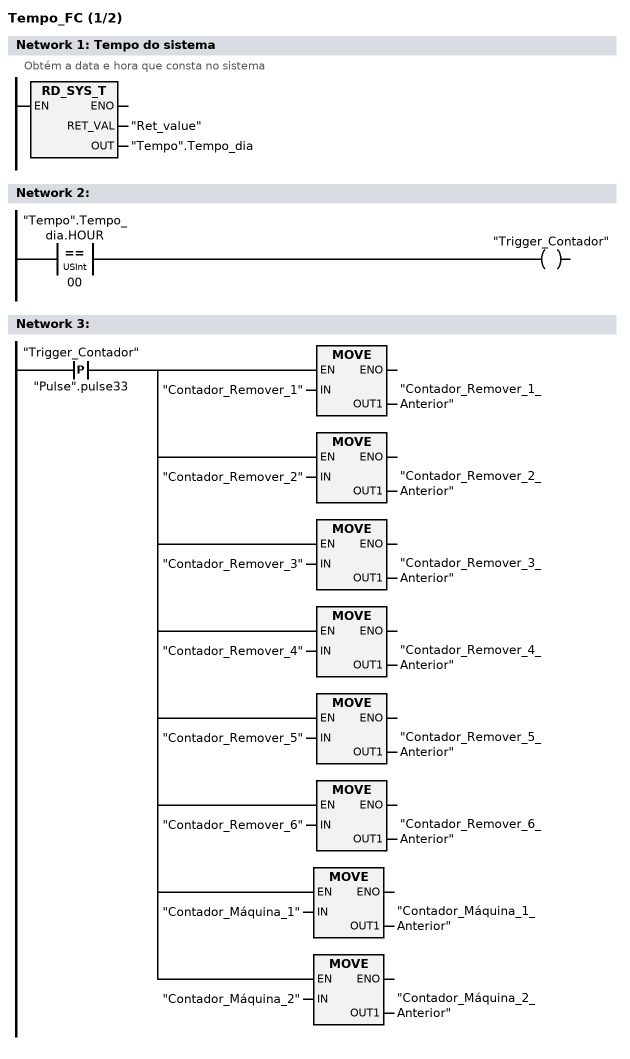
   "Ret_value" := RD_SYS_T(OUT => "Tempo".Tempo_dia);
END_REGION

REGION Network 2
   RUNG wire#powerrail
      { S7_Templates := "SrcType := USInt" } EQ_Contact(in1 := "Tempo".Tempo_dia.HOUR, in2 := 00)
      Coil( "Trigger_Contador" )
   END_RUNG
   // the same network as SCL:
   "Trigger_Contador" := "Tempo".Tempo_dia.HOUR = 00;
END_REGION

REGION Network 3
   RUNG wire#powerrail
      P_Contact(operand := "Trigger_Contador", bit := "Pulse".pulse33)
      wire#w1
      Move(in := "Contador_Remover_1", out1 => "Contador_Remover_1_Anterior")
   END_RUNG
   RUNG wire#w1
      Move(in := "Contador_Remover_2", out1 => "Contador_Remover_2_Anterior")
   END_RUNG
   RUNG wire#w1
      Move(in := "Contador_Remover_3", out1 => "Contador_Remover_3_Anterior")
   END_RUNG
   RUNG wire#w1
      Move(in := "Contador_Remover_4", out1 => "Contador_Remover_4_Anterior")
   END_RUNG
   RUNG wire#w1
      Move(in := "Contador_Remover_5", out1 => "Contador_Remover_5_Anterior")
   END_RUNG
   RUNG wire#w1
      Move(in := "Contador_Remover_6", out1 => "Contador_Remover_6_Anterior")
   END_RUNG
   RUNG wire#w1
      Move(in := "Contador_Máquina_1", out1 => "Contador_Máquina_1_Anterior")
   END_RUNG
   RUNG wire#w1
      Move(in := "Contador_Máquina_2", out1 => "Contador_Máquina_2_Anterior")
   END_RUNG
   // the same network as SCL:
   #_w1 := "Trigger_Contador" AND NOT "Pulse".pulse33;   // rising edge of "Trigger_Contador"
   "Pulse".pulse33 := "Trigger_Contador";
   IF #_w1 THEN
       "Contador_Remover_1_Anterior" := "Contador_Remover_1";
       "Contador_Remover_2_Anterior" := "Contador_Remover_2";
       "Contador_Remover_3_Anterior" := "Contador_Remover_3";
       "Contador_Remover_4_Anterior" := "Contador_Remover_4";
       "Contador_Remover_5_Anterior" := "Contador_Remover_5";
       "Contador_Remover_6_Anterior" := "Contador_Remover_6";
       "Contador_Máquina_1_Anterior" := "Contador_Máquina_1";
       "Contador_Máquina_2_Anterior" := "Contador_Máquina_2";
   END_IF;
END_REGION

REGION Network 4: Reset de contadores
   // Reset diário de todos os contadores, à meia-noite
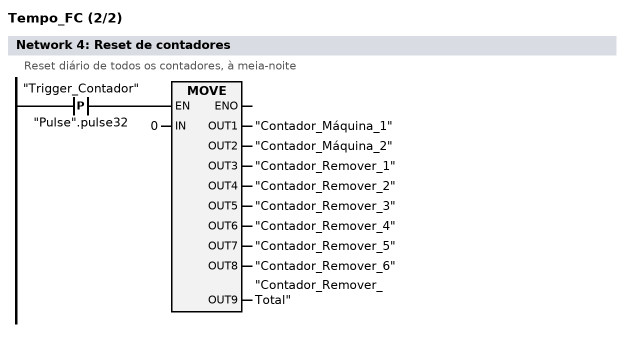
   RUNG wire#powerrail
      P_Contact(operand := "Trigger_Contador", bit := "Pulse".pulse32)
      Move(in := 0, out1 => "Contador_Máquina_1", out2 => "Contador_Máquina_2", out3 => "Contador_Remover_1", out4 => "Contador_Remover_2", out5 => "Contador_Remover_3", out6 => "Contador_Remover_4", out7 => "Contador_Remover_5", out8 => "Contador_Remover_6", out9 => "Contador_Remover_Total")
   END_RUNG
   // the same network as SCL:
   #_w1 := "Trigger_Contador" AND NOT "Pulse".pulse32;   // rising edge of "Trigger_Contador"
   "Pulse".pulse32 := "Trigger_Contador";
   IF #_w1 THEN
       "Contador_Máquina_1" := 0;
       "Contador_Máquina_2" := 0;
       "Contador_Remover_1" := 0;
       "Contador_Remover_2" := 0;
       "Contador_Remover_3" := 0;
       "Contador_Remover_4" := 0;
       "Contador_Remover_5" := 0;
       "Contador_Remover_6" := 0;
       "Contador_Remover_Total" := 0;
   END_IF;
END_REGION
END_FUNCTION

FUNCTION "MoveToSendData_PLC1" : Void   // FC10, SCL
{ S7_Optimized_Access := 'TRUE' }
VERSION : 0.1
   VAR_INPUT
      Contador_Remover_1 : DWord;
      Contador_Remover_2 : DWord;
      Contador_Remover_3 : DWord;
      Contador_Remover_4 : DWord;
      Contador_Remover_5 : DWord;
      Contador_Remover_6 : DWord;
      Contador_Remover_Total : DWord;
      Contador_Máquina_1 : DWord;
      Contador_Máquina_2 : DWord;
      "Valvula Enchimento Tanque 1" : Real;
      "Valvula Descarga Tanque 1" : Real;
      "Valvula Enchimento Tanque 2" : Real;
      "Valvula Descarga Tanque 2" : Real;
      Nivel_1_convertido_Scada : Real;
      Nivel_2_convertido_Scada : Real;
      Aviso_Nenhuma_Máquina_Habilitada : Bool;
      Aviso_Nenhum_Remover_Habilitado : Bool;
      Aviso_Sem_Condições_Empilhar : Bool;
      Set_vel_T3 : Real;
      Set_vel_T4 : Real;
      Set_vel_T5 : Real;
      Set_vel_T6 : Real;
      Set_vel_T7 : Real;
   END_VAR
   VAR_OUTPUT
      OUT_Contador_Remover_1 : DWord;
      OUT_Contador_Remover_2 : DWord;
      OUT_Contador_Remover_3 : DWord;
      OUT_Contador_Remover_4 : DWord;
      OUT_Contador_Remover_5 : DWord;
      OUT_Contador_Remover_6 : DWord;
      OUT_Contador_Remover_Total : DWord;
      OUT_Contador_Máquina_1 : DWord;
      OUT_Contador_Máquina_2 : DWord;
      "OUT_Valvula Enchimento Tanque 1" : Real;
      "OUT_Valvula Descarga Tanque 1" : Real;
      "OUT_Valvula Enchimento Tanque 2" : Real;
      "OUT_Valvula Descarga Tanque 2" : Real;
      OUT_Nivel_1_convertido_Scada : Real;
      OUT_Nivel_2_convertido_Scada : Real;
      OUT_Aviso_Nenhuma_Máquina_Habilitada : Bool;
      OUT_Aviso_Nenhum_Remover_Habilitado : Bool;
      OUT_Aviso_Sem_Condições_Empilhar : Bool;
      OUT_Set_vel_T3 : Real;
      OUT_Set_vel_T4 : Real;
      OUT_Set_vel_T5 : Real;
      OUT_Set_vel_T6 : Real;
      OUT_Set_vel_T7 : Real;
   END_VAR
BEGIN


           #OUT_Contador_Remover_1 := #Contador_Remover_1;
           #OUT_Contador_Remover_2 := #Contador_Remover_2;
           #OUT_Contador_Remover_3 := #Contador_Remover_3;
           #OUT_Contador_Remover_4 := #Contador_Remover_4;
           #OUT_Contador_Remover_5 := #Contador_Remover_5;
           #OUT_Contador_Remover_6 := #Contador_Remover_6;
           #OUT_Contador_Remover_Total := #Contador_Remover_Total;
           #OUT_Contador_Máquina_1 := #Contador_Máquina_1;
           #OUT_Contador_Máquina_2 := #Contador_Máquina_2;

           #"OUT_Valvula Enchimento Tanque 1" := #"Valvula Enchimento Tanque 1";
           #"OUT_Valvula Descarga Tanque 1":= #"Valvula Descarga Tanque 1";
           #"OUT_Valvula Enchimento Tanque 2" := #"Valvula Enchimento Tanque 2";
           #"OUT_Valvula Descarga Tanque 2":= #"Valvula Descarga Tanque 2";

           #OUT_Nivel_1_convertido_Scada := #Nivel_1_convertido_Scada;
           #OUT_Nivel_2_convertido_Scada := #Nivel_2_convertido_Scada;

           #OUT_Aviso_Nenhuma_Máquina_Habilitada := #Aviso_Nenhuma_Máquina_Habilitada;
           #OUT_Aviso_Nenhum_Remover_Habilitado := #Aviso_Nenhum_Remover_Habilitado;
           #OUT_Aviso_Sem_Condições_Empilhar := #Aviso_Sem_Condições_Empilhar;


           #OUT_Set_vel_T3 := #Set_vel_T3;
           #OUT_Set_vel_T4 := #Set_vel_T4;
           #OUT_Set_vel_T5 := #Set_vel_T5;
           #OUT_Set_vel_T6 := #Set_vel_T6;
           #OUT_Set_vel_T7 := #Set_vel_T7;
END_FUNCTION

FUNCTION "MoveToReceiveData_PLC1" : Void   // FC11, SCL
{ S7_Optimized_Access := 'TRUE' }
VERSION : 0.1
   VAR_INPUT
      Start : Bool;
      Stop : Bool;
      Emergência : Bool;
      Habilita_Remover_1 : Bool;
      Habilita_Remover_2 : Bool;
      Habilita_Remover_3 : Bool;
      Habilita_Remover_4 : Bool;
      Habilita_Remover_5 : Bool;
      Habilita_Remover_6 : Bool;
      Habilita_Máquina_1 : Bool;
      Habilita_Máquina_2 : Bool;
      Empilhar : Bool;
      Reset_Cont_Diario : DWord;
      "Reset Contadores Maquinas" : Bool;
      "Reset Contadores Postos" : Bool;
      Máquina2_Tampas : Bool;
      Máquina1_Tampas : Bool;
   END_VAR
   VAR_OUTPUT
      OUT_Start : Bool;
      OUT_Stop : Bool;
      OUT_Emergência : Bool;
      OUT_Habilita_Remover_1 : Bool;
      OUT_Habilita_Remover_2 : Bool;
      OUT_Habilita_Remover_3 : Bool;
      OUT_Habilita_Remover_4 : Bool;
      OUT_Habilita_Remover_5 : Bool;
      OUT_Habilita_Remover_6 : Bool;
      OUT_Habilita_Máquina_1 : Bool;
      OUT_Habilita_Máquina_2 : Bool;
      OUT_Empilhar : Bool;
      OUT_Reset_Cont_Diario : DWord;
      "OUT_Reset Contadores Maquinas" : Bool;
      "OUT_Reset Contadores Postos" : Bool;
      OUT_Máquina2_Tampas : Bool;
      OUT_Máquina1_Tampas : Bool;
   END_VAR
BEGIN



       #OUT_Start := #Start;
       #OUT_Stop := #Stop;
       #"OUT_Emergência" := #"Emergência";

       #OUT_Habilita_Remover_1 := #Habilita_Remover_1;
       #OUT_Habilita_Remover_2 := #Habilita_Remover_2;
       #OUT_Habilita_Remover_3 := #Habilita_Remover_3;
       #OUT_Habilita_Remover_4 := #Habilita_Remover_4;
       #OUT_Habilita_Remover_5 := #Habilita_Remover_5;
       #OUT_Habilita_Remover_6 := #Habilita_Remover_6;

       #"OUT_Habilita_Máquina_1" := #"Habilita_Máquina_1";
       #"OUT_Habilita_Máquina_2" := #"Habilita_Máquina_2";

       #OUT_Empilhar := #Empilhar;

       #OUT_Reset_Cont_Diario := #Reset_Cont_Diario;
       #"OUT_Reset Contadores Maquinas" := #"Reset Contadores Maquinas";
       #"OUT_Reset Contadores Postos" := #"Reset Contadores Postos";

       #OUT_Máquina2_Tampas := #Máquina2_Tampas;
       #OUT_Máquina1_Tampas := #Máquina1_Tampas;
END_FUNCTION

ORGANIZATION_BLOCK "Main"   // OB1, LAD, ProgramCycle
TITLE = "Main Program Sweep (Cycle)"
{ S7_Optimized_Access := 'TRUE' }
VERSION : 0.1
   VAR_INPUT
      Initial_Call : Bool;   // Initial call of this OB
      Remanence : Bool;   // =True, if remanent data are available
   END_VAR
   VAR_TEMP   // added for the SCL form of the ladder/FBD networks
      _w1 : Bool;
   END_VAR
BEGIN

REGION Network 1: Inicialização
   // Dá set ao bit do botão de stop para simular o botão de stop NC.
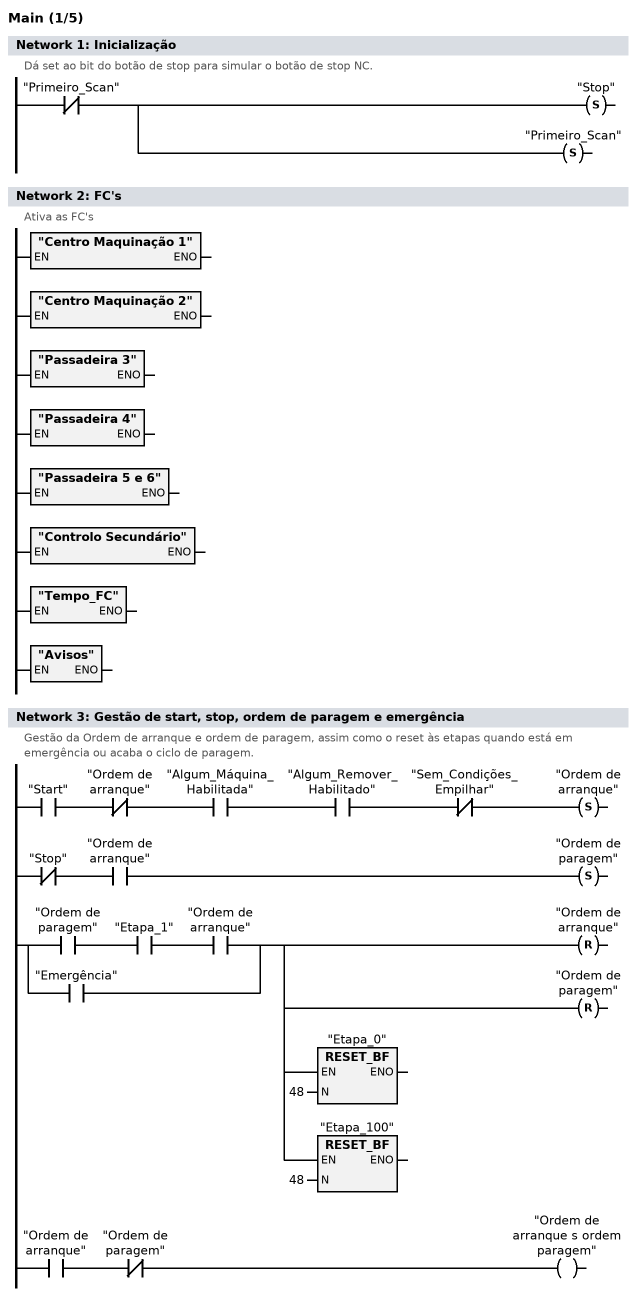
   RUNG wire#powerrail
      I_Contact( "Primeiro_Scan" )
      wire#w1
      S_Coil( "Stop" )
   END_RUNG
   RUNG wire#w1
      S_Coil( "Primeiro_Scan" )
   END_RUNG
   // the same network as SCL:
   IF NOT "Primeiro_Scan" THEN
       "Stop" := TRUE;
       "Primeiro_Scan" := TRUE;
   END_IF;
END_REGION

REGION Network 2: FC's
   // Ativa as FC's
   RUNG wire#powerrail
      "Centro Maquinação 1"()
   END_RUNG
   RUNG wire#powerrail
      "Centro Maquinação 2"()
   END_RUNG
   RUNG wire#powerrail
      "Passadeira 3"()
   END_RUNG
   RUNG wire#powerrail
      "Passadeira 4"()
   END_RUNG
   RUNG wire#powerrail
      "Passadeira 5 e 6"()
   END_RUNG
   RUNG wire#powerrail
      "Controlo Secundário"()
   END_RUNG
   RUNG wire#powerrail
      "Tempo_FC"()
   END_RUNG
   RUNG wire#powerrail
      "Avisos"()
   END_RUNG
   // the same network as SCL:
   "Centro Maquinação 1"();
   "Centro Maquinação 2"();
   "Passadeira 3"();
   "Passadeira 4"();
   "Passadeira 5 e 6"();
   "Controlo Secundário"();
   "Tempo_FC"();
   "Avisos"();
END_REGION

REGION Network 3: Gestão de start, stop, ordem de paragem e emergência
   // Gestão da Ordem de arranque e ordem de paragem, assim como o reset às etapas quando está em emergência ou acaba o ciclo de paragem.
   // no SCL statement known for RBitfield: written as a call
   IF "Start" AND NOT "Ordem de arranque" AND "Algum_Máquina_Habilitada" AND "Algum_Remover_Habilitado" AND NOT "Sem_Condições_Empilhar" THEN
       "Ordem de arranque" := TRUE;
   END_IF;
   IF NOT "Stop" AND "Ordem de arranque" THEN "Ordem de paragem" := TRUE; END_IF;
   #_w1 := ("Ordem de paragem" AND "Etapa_1" AND "Ordem de arranque") OR "Emergência";
   IF #_w1 THEN
       "Ordem de arranque" := FALSE;
       "Ordem de paragem" := FALSE;
       RESET_BF(operand := "Etapa_0", n := 48);
       RESET_BF(operand := "Etapa_100", n := 48);
   END_IF;
   "Ordem de arranque s ordem paragem" := "Ordem de arranque" AND NOT "Ordem de paragem";
END_REGION

REGION Network 4: Ordem de arranque
   // No pulse da ordem de arranque dá set à etapa 0 para iniciar
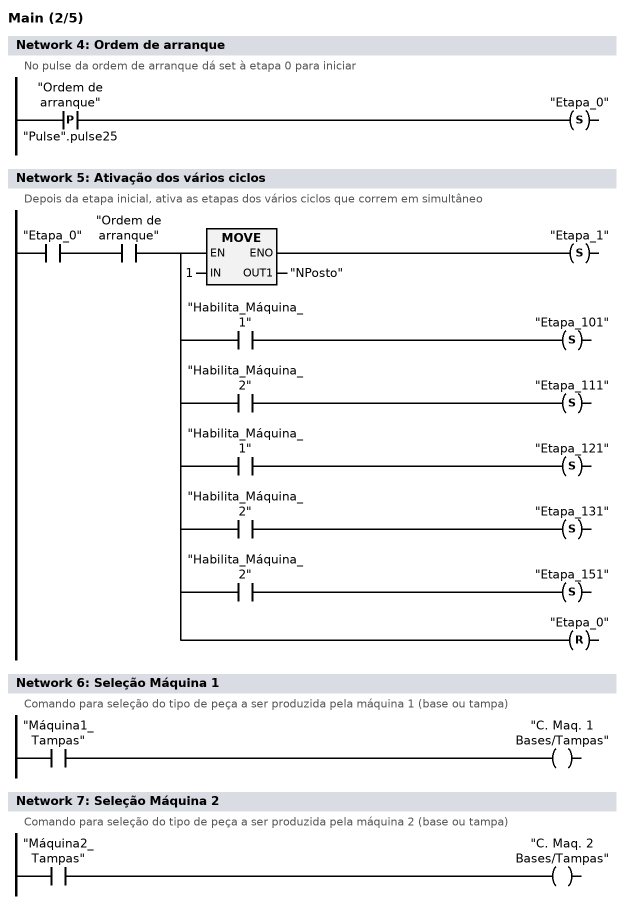
   RUNG wire#powerrail
      P_Contact(operand := "Ordem de arranque", bit := "Pulse".pulse25)
      S_Coil( "Etapa_0" )
   END_RUNG
   // the same network as SCL:
   #_w1 := "Ordem de arranque" AND NOT "Pulse".pulse25;   // rising edge of "Ordem de arranque"
   "Pulse".pulse25 := "Ordem de arranque";
   IF #_w1 THEN "Etapa_0" := TRUE; END_IF;
END_REGION

REGION Network 5: Ativação dos vários ciclos
   // Depois da etapa inicial, ativa as etapas dos vários ciclos que correm em simultâneo
   RUNG wire#powerrail
      Contact( "Etapa_0" )
      Contact( "Ordem de arranque" )
      wire#w1
      Move(in := 1, out1 => "NPosto")
      S_Coil( "Etapa_1" )
   END_RUNG
   RUNG wire#w1
      Contact( "Habilita_Máquina_1" )
      S_Coil( "Etapa_101" )
   END_RUNG
   RUNG wire#w1
      Contact( "Habilita_Máquina_2" )
      S_Coil( "Etapa_111" )
   END_RUNG
   RUNG wire#w1
      Contact( "Habilita_Máquina_1" )
      S_Coil( "Etapa_121" )
   END_RUNG
   RUNG wire#w1
      Contact( "Habilita_Máquina_2" )
      S_Coil( "Etapa_131" )
   END_RUNG
   RUNG wire#w1
      Contact( "Habilita_Máquina_2" )
      S_Coil( "Etapa_151" )
   END_RUNG
   RUNG wire#w1
      R_Coil( "Etapa_0" )
   END_RUNG
   // the same network as SCL:
   #_w1 := "Etapa_0" AND "Ordem de arranque";
   IF #_w1 THEN
       "NPosto" := 1;
       "Etapa_1" := TRUE;
   END_IF;
   IF #_w1 AND "Habilita_Máquina_1" THEN "Etapa_101" := TRUE; END_IF;
   IF #_w1 AND "Habilita_Máquina_2" THEN "Etapa_111" := TRUE; END_IF;
   IF #_w1 AND "Habilita_Máquina_1" THEN "Etapa_121" := TRUE; END_IF;
   IF #_w1 AND "Habilita_Máquina_2" THEN
       "Etapa_131" := TRUE;
       "Etapa_151" := TRUE;
   END_IF;
   IF #_w1 THEN "Etapa_0" := FALSE; END_IF;
END_REGION

REGION Network 6: Seleção Máquina 1
   // Comando para seleção do tipo de peça a ser produzida pela máquina 1 (base ou tampa)
   RUNG wire#powerrail
      Contact( "Máquina1_Tampas" )
      Coil( "C. Maq. 1 Bases/Tampas" )
   END_RUNG
   // the same network as SCL:
   "C. Maq. 1 Bases/Tampas" := "Máquina1_Tampas";
END_REGION

REGION Network 7: Seleção Máquina 2
   // Comando para seleção do tipo de peça a ser produzida pela máquina 2 (base ou tampa)
   RUNG wire#powerrail
      Contact( "Máquina2_Tampas" )
      Coil( "C. Maq. 2 Bases/Tampas" )
   END_RUNG
   // the same network as SCL:
   "C. Maq. 2 Bases/Tampas" := "Máquina2_Tampas";
END_REGION

REGION Network 8: Verificação de postos habilitados
   // Verificação de que algum posto de armazenamento está habilitado
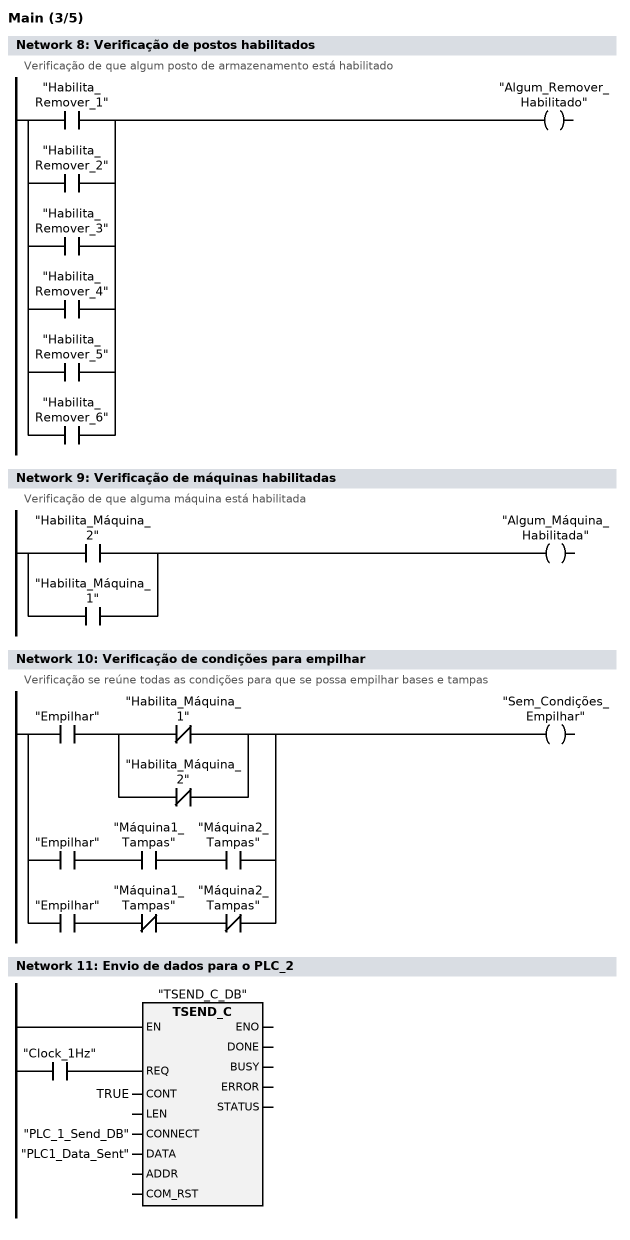
   RUNG wire#powerrail
      Contact( "Habilita_Remover_1" )
      wire#w1
      Coil( "Algum_Remover_Habilitado" )
   END_RUNG
   RUNG wire#powerrail
      Contact( "Habilita_Remover_2" )
   END_RUNG wire#w1
   RUNG wire#powerrail
      Contact( "Habilita_Remover_3" )
   END_RUNG wire#w1
   RUNG wire#powerrail
      Contact( "Habilita_Remover_4" )
   END_RUNG wire#w1
   RUNG wire#powerrail
      Contact( "Habilita_Remover_5" )
   END_RUNG wire#w1
   RUNG wire#powerrail
      Contact( "Habilita_Remover_6" )
   END_RUNG wire#w1
   // the same network as SCL:
   "Algum_Remover_Habilitado" := "Habilita_Remover_1" OR "Habilita_Remover_2" OR "Habilita_Remover_3" OR "Habilita_Remover_4" OR "Habilita_Remover_5" OR "Habilita_Remover_6";
END_REGION

REGION Network 9: Verificação de máquinas habilitadas
   // Verificação de que alguma máquina está habilitada
   RUNG wire#powerrail
      Contact( "Habilita_Máquina_2" )
      wire#w1
      Coil( "Algum_Máquina_Habilitada" )
   END_RUNG
   RUNG wire#powerrail
      Contact( "Habilita_Máquina_1" )
   END_RUNG wire#w1
   // the same network as SCL:
   "Algum_Máquina_Habilitada" := "Habilita_Máquina_2" OR "Habilita_Máquina_1";
END_REGION

REGION Network 10: Verificação de condições para empilhar
   // Verificação se reúne todas as condições para que se possa empilhar bases e tampas
   RUNG wire#powerrail
      Contact( "Empilhar" )
      wire#w1
      I_Contact( "Habilita_Máquina_1" )
      wire#w2
      Coil( "Sem_Condições_Empilhar" )
   END_RUNG
   RUNG wire#w1
      I_Contact( "Habilita_Máquina_2" )
   END_RUNG wire#w2
   RUNG wire#powerrail
      Contact( "Empilhar" )
      Contact( "Máquina1_Tampas" )
      Contact( "Máquina2_Tampas" )
   END_RUNG wire#w2
   RUNG wire#powerrail
      Contact( "Empilhar" )
      I_Contact( "Máquina1_Tampas" )
      I_Contact( "Máquina2_Tampas" )
   END_RUNG wire#w2
   // the same network as SCL:
   "Sem_Condições_Empilhar" := ("Empilhar" AND (NOT "Habilita_Máquina_1" OR NOT "Habilita_Máquina_2")) OR ("Empilhar" AND "Máquina1_Tampas" AND "Máquina2_Tampas") OR ("Empilhar" AND NOT "Máquina1_Tampas" AND NOT "Máquina2_Tampas");
END_REGION

REGION Network 11: Envio de dados para o PLC_2
   "TSEND_C_DB"(REQ := "Clock_1Hz", CONT := TRUE, CONNECT := "PLC_1_Send_DB", DATA := "PLC1_Data_Sent");   // TSEND_C
END_REGION

REGION Network 12: Função para copiar os valores das variáveis para uma DB que partilhará os dados com o PLC_2
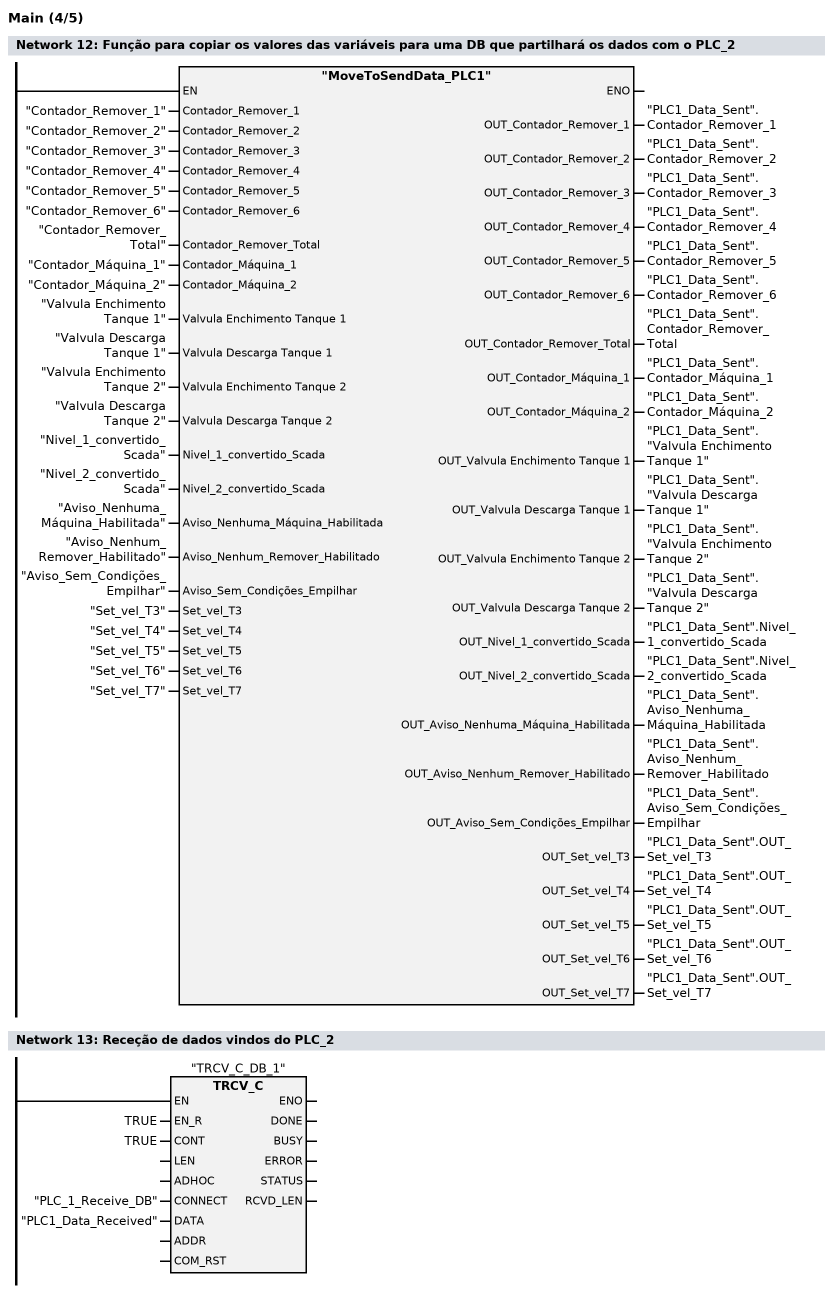
   RUNG wire#powerrail
      "MoveToSendData_PLC1"(Contador_Remover_1 := "Contador_Remover_1", Contador_Remover_2 := "Contador_Remover_2", Contador_Remover_3 := "Contador_Remover_3", Contador_Remover_4 := "Contador_Remover_4", Contador_Remover_5 := "Contador_Remover_5", Contador_Remover_6 := "Contador_Remover_6", Contador_Remover_Total := "Contador_Remover_Total", Contador_Máquina_1 := "Contador_Máquina_1", Contador_Máquina_2 := "Contador_Máquina_2", "Valvula Enchimento Tanque 1" := "Valvula Enchimento Tanque 1", "Valvula Descarga Tanque 1" := "Valvula Descarga Tanque 1", "Valvula Enchimento Tanque 2" := "Valvula Enchimento Tanque 2", "Valvula Descarga Tanque 2" := "Valvula Descarga Tanque 2", Nivel_1_convertido_Scada := "Nivel_1_convertido_Scada", Nivel_2_convertido_Scada := "Nivel_2_convertido_Scada", Aviso_Nenhuma_Máquina_Habilitada := "Aviso_Nenhuma_Máquina_Habilitada", Aviso_Nenhum_Remover_Habilitado := "Aviso_Nenhum_Remover_Habilitado", Aviso_Sem_Condições_Empilhar := "Aviso_Sem_Condições_Empilhar", Set_vel_T3 := "Set_vel_T3", Set_vel_T4 := "Set_vel_T4", Set_vel_T5 := "Set_vel_T5", Set_vel_T6 := "Set_vel_T6", Set_vel_T7 := "Set_vel_T7", OUT_Contador_Remover_1 => "PLC1_Data_Sent".Contador_Remover_1, OUT_Contador_Remover_2 => "PLC1_Data_Sent".Contador_Remover_2, OUT_Contador_Remover_3 => "PLC1_Data_Sent".Contador_Remover_3, OUT_Contador_Remover_4 => "PLC1_Data_Sent".Contador_Remover_4, OUT_Contador_Remover_5 => "PLC1_Data_Sent".Contador_Remover_5, OUT_Contador_Remover_6 => "PLC1_Data_Sent".Contador_Remover_6, OUT_Contador_Remover_Total => "PLC1_Data_Sent".Contador_Remover_Total, OUT_Contador_Máquina_1 => "PLC1_Data_Sent".Contador_Máquina_1, OUT_Contador_Máquina_2 => "PLC1_Data_Sent".Contador_Máquina_2, "OUT_Valvula Enchimento Tanque 1" => "PLC1_Data_Sent"."Valvula Enchimento Tanque 1", "OUT_Valvula Descarga Tanque 1" => "PLC1_Data_Sent"."Valvula Descarga Tanque 1", "OUT_Valvula Enchimento Tanque 2" => "PLC1_Data_Sent"."Valvula Enchimento Tanque 2", "OUT_Valvula Descarga Tanque 2" => "PLC1_Data_Sent"."Valvula Descarga Tanque 2", OUT_Nivel_1_convertido_Scada => "PLC1_Data_Sent".Nivel_1_convertido_Scada, OUT_Nivel_2_convertido_Scada => "PLC1_Data_Sent".Nivel_2_convertido_Scada, OUT_Aviso_Nenhuma_Máquina_Habilitada => "PLC1_Data_Sent".Aviso_Nenhuma_Máquina_Habilitada, OUT_Aviso_Nenhum_Remover_Habilitado => "PLC1_Data_Sent".Aviso_Nenhum_Remover_Habilitado, OUT_Aviso_Sem_Condições_Empilhar => "PLC1_Data_Sent".Aviso_Sem_Condições_Empilhar, OUT_Set_vel_T3 => "PLC1_Data_Sent".OUT_Set_vel_T3, OUT_Set_vel_T4 => "PLC1_Data_Sent".OUT_Set_vel_T4, OUT_Set_vel_T5 => "PLC1_Data_Sent".OUT_Set_vel_T5, OUT_Set_vel_T6 => "PLC1_Data_Sent".OUT_Set_vel_T6, OUT_Set_vel_T7 => "PLC1_Data_Sent".OUT_Set_vel_T7)
   END_RUNG
   // the same network as SCL:
   "MoveToSendData_PLC1"(Contador_Remover_1 := "Contador_Remover_1",
                         Contador_Remover_2 := "Contador_Remover_2",
                         Contador_Remover_3 := "Contador_Remover_3",
                         Contador_Remover_4 := "Contador_Remover_4",
                         Contador_Remover_5 := "Contador_Remover_5",
                         Contador_Remover_6 := "Contador_Remover_6",
                         Contador_Remover_Total := "Contador_Remover_Total",
                         Contador_Máquina_1 := "Contador_Máquina_1",
                         Contador_Máquina_2 := "Contador_Máquina_2",
                         "Valvula Enchimento Tanque 1" := "Valvula Enchimento Tanque 1",
                         "Valvula Descarga Tanque 1" := "Valvula Descarga Tanque 1",
                         "Valvula Enchimento Tanque 2" := "Valvula Enchimento Tanque 2",
                         "Valvula Descarga Tanque 2" := "Valvula Descarga Tanque 2",
                         Nivel_1_convertido_Scada := "Nivel_1_convertido_Scada",
                         Nivel_2_convertido_Scada := "Nivel_2_convertido_Scada",
                         Aviso_Nenhuma_Máquina_Habilitada := "Aviso_Nenhuma_Máquina_Habilitada",
                         Aviso_Nenhum_Remover_Habilitado := "Aviso_Nenhum_Remover_Habilitado",
                         Aviso_Sem_Condições_Empilhar := "Aviso_Sem_Condições_Empilhar",
                         Set_vel_T3 := "Set_vel_T3",
                         Set_vel_T4 := "Set_vel_T4",
                         Set_vel_T5 := "Set_vel_T5",
                         Set_vel_T6 := "Set_vel_T6",
                         Set_vel_T7 := "Set_vel_T7",
                         OUT_Contador_Remover_1 => "PLC1_Data_Sent".Contador_Remover_1,
                         OUT_Contador_Remover_2 => "PLC1_Data_Sent".Contador_Remover_2,
                         OUT_Contador_Remover_3 => "PLC1_Data_Sent".Contador_Remover_3,
                         OUT_Contador_Remover_4 => "PLC1_Data_Sent".Contador_Remover_4,
                         OUT_Contador_Remover_5 => "PLC1_Data_Sent".Contador_Remover_5,
                         OUT_Contador_Remover_6 => "PLC1_Data_Sent".Contador_Remover_6,
                         OUT_Contador_Remover_Total => "PLC1_Data_Sent".Contador_Remover_Total,
                         OUT_Contador_Máquina_1 => "PLC1_Data_Sent".Contador_Máquina_1,
                         OUT_Contador_Máquina_2 => "PLC1_Data_Sent".Contador_Máquina_2,
                         "OUT_Valvula Enchimento Tanque 1" => "PLC1_Data_Sent"."Valvula Enchimento Tanque 1",
                         "OUT_Valvula Descarga Tanque 1" => "PLC1_Data_Sent"."Valvula Descarga Tanque 1",
                         "OUT_Valvula Enchimento Tanque 2" => "PLC1_Data_Sent"."Valvula Enchimento Tanque 2",
                         "OUT_Valvula Descarga Tanque 2" => "PLC1_Data_Sent"."Valvula Descarga Tanque 2",
                         OUT_Nivel_1_convertido_Scada => "PLC1_Data_Sent".Nivel_1_convertido_Scada,
                         OUT_Nivel_2_convertido_Scada => "PLC1_Data_Sent".Nivel_2_convertido_Scada,
                         OUT_Aviso_Nenhuma_Máquina_Habilitada => "PLC1_Data_Sent".Aviso_Nenhuma_Máquina_Habilitada,
                         OUT_Aviso_Nenhum_Remover_Habilitado => "PLC1_Data_Sent".Aviso_Nenhum_Remover_Habilitado,
                         OUT_Aviso_Sem_Condições_Empilhar => "PLC1_Data_Sent".Aviso_Sem_Condições_Empilhar,
                         OUT_Set_vel_T3 => "PLC1_Data_Sent".OUT_Set_vel_T3,
                         OUT_Set_vel_T4 => "PLC1_Data_Sent".OUT_Set_vel_T4,
                         OUT_Set_vel_T5 => "PLC1_Data_Sent".OUT_Set_vel_T5,
                         OUT_Set_vel_T6 => "PLC1_Data_Sent".OUT_Set_vel_T6,
                         OUT_Set_vel_T7 => "PLC1_Data_Sent".OUT_Set_vel_T7);
END_REGION

REGION Network 13: Receção de dados vindos do PLC_2
   "TRCV_C_DB_1"(EN_R := TRUE, CONT := TRUE, CONNECT := "PLC_1_Receive_DB", DATA := "PLC1_Data_Received");   // TRCV_C
END_REGION

REGION Network 14
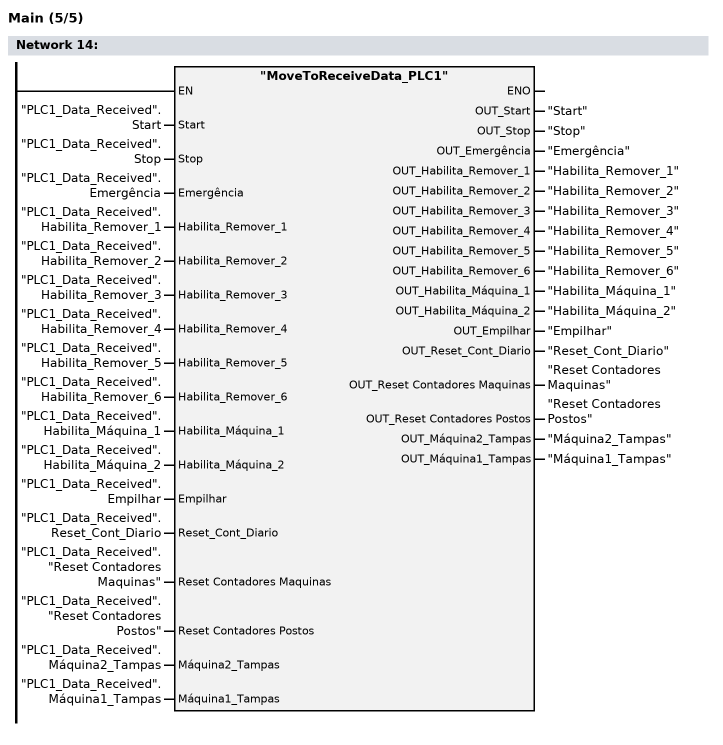
   RUNG wire#powerrail
      "MoveToReceiveData_PLC1"(Start := "PLC1_Data_Received".Start, Stop := "PLC1_Data_Received".Stop, Emergência := "PLC1_Data_Received".Emergência, Habilita_Remover_1 := "PLC1_Data_Received".Habilita_Remover_1, Habilita_Remover_2 := "PLC1_Data_Received".Habilita_Remover_2, Habilita_Remover_3 := "PLC1_Data_Received".Habilita_Remover_3, Habilita_Remover_4 := "PLC1_Data_Received".Habilita_Remover_4, Habilita_Remover_5 := "PLC1_Data_Received".Habilita_Remover_5, Habilita_Remover_6 := "PLC1_Data_Received".Habilita_Remover_6, Habilita_Máquina_1 := "PLC1_Data_Received".Habilita_Máquina_1, Habilita_Máquina_2 := "PLC1_Data_Received".Habilita_Máquina_2, Empilhar := "PLC1_Data_Received".Empilhar, Reset_Cont_Diario := "PLC1_Data_Received".Reset_Cont_Diario, "Reset Contadores Maquinas" := "PLC1_Data_Received"."Reset Contadores Maquinas", "Reset Contadores Postos" := "PLC1_Data_Received"."Reset Contadores Postos", Máquina2_Tampas := "PLC1_Data_Received".Máquina2_Tampas, Máquina1_Tampas := "PLC1_Data_Received".Máquina1_Tampas, OUT_Start => "Start", OUT_Stop => "Stop", OUT_Emergência => "Emergência", OUT_Habilita_Remover_1 => "Habilita_Remover_1", OUT_Habilita_Remover_2 => "Habilita_Remover_2", OUT_Habilita_Remover_3 => "Habilita_Remover_3", OUT_Habilita_Remover_4 => "Habilita_Remover_4", OUT_Habilita_Remover_5 => "Habilita_Remover_5", OUT_Habilita_Remover_6 => "Habilita_Remover_6", OUT_Habilita_Máquina_1 => "Habilita_Máquina_1", OUT_Habilita_Máquina_2 => "Habilita_Máquina_2", OUT_Empilhar => "Empilhar", OUT_Reset_Cont_Diario => "Reset_Cont_Diario", "OUT_Reset Contadores Maquinas" => "Reset Contadores Maquinas", "OUT_Reset Contadores Postos" => "Reset Contadores Postos", OUT_Máquina2_Tampas => "Máquina2_Tampas", OUT_Máquina1_Tampas => "Máquina1_Tampas")
   END_RUNG
   // the same network as SCL:
   "MoveToReceiveData_PLC1"(Start := "PLC1_Data_Received".Start,
                           Stop := "PLC1_Data_Received".Stop,
                           Emergência := "PLC1_Data_Received".Emergência,
                           Habilita_Remover_1 := "PLC1_Data_Received".Habilita_Remover_1,
                           Habilita_Remover_2 := "PLC1_Data_Received".Habilita_Remover_2,
                           Habilita_Remover_3 := "PLC1_Data_Received".Habilita_Remover_3,
                           Habilita_Remover_4 := "PLC1_Data_Received".Habilita_Remover_4,
                           Habilita_Remover_5 := "PLC1_Data_Received".Habilita_Remover_5,
                           Habilita_Remover_6 := "PLC1_Data_Received".Habilita_Remover_6,
                           Habilita_Máquina_1 := "PLC1_Data_Received".Habilita_Máquina_1,
                           Habilita_Máquina_2 := "PLC1_Data_Received".Habilita_Máquina_2,
                           Empilhar := "PLC1_Data_Received".Empilhar,
                           Reset_Cont_Diario := "PLC1_Data_Received".Reset_Cont_Diario,
                           "Reset Contadores Maquinas" := "PLC1_Data_Received"."Reset Contadores Maquinas",
                           "Reset Contadores Postos" := "PLC1_Data_Received"."Reset Contadores Postos",
                           Máquina2_Tampas := "PLC1_Data_Received".Máquina2_Tampas,
                           Máquina1_Tampas := "PLC1_Data_Received".Máquina1_Tampas,
                           OUT_Start => "Start",
                           OUT_Stop => "Stop",
                           OUT_Emergência => "Emergência",
                           OUT_Habilita_Remover_1 => "Habilita_Remover_1",
                           OUT_Habilita_Remover_2 => "Habilita_Remover_2",
                           OUT_Habilita_Remover_3 => "Habilita_Remover_3",
                           OUT_Habilita_Remover_4 => "Habilita_Remover_4",
                           OUT_Habilita_Remover_5 => "Habilita_Remover_5",
                           OUT_Habilita_Remover_6 => "Habilita_Remover_6",
                           OUT_Habilita_Máquina_1 => "Habilita_Máquina_1",
                           OUT_Habilita_Máquina_2 => "Habilita_Máquina_2",
                           OUT_Empilhar => "Empilhar",
                           OUT_Reset_Cont_Diario => "Reset_Cont_Diario",
                           "OUT_Reset Contadores Maquinas" => "Reset Contadores Maquinas",
                           "OUT_Reset Contadores Postos" => "Reset Contadores Postos",
                           OUT_Máquina2_Tampas => "Máquina2_Tampas",
                           OUT_Máquina1_Tampas => "Máquina1_Tampas");
END_REGION
END_ORGANIZATION_BLOCK

ORGANIZATION_BLOCK "Cyclic interrupt"   // OB30, LAD, CyclicInterrupt
TITLE = PID Tanque 1
{ S7_Optimized_Access := 'TRUE' }
VERSION : 0.1
   VAR_INPUT
      Initial_Call : Bool;   // Initial call of this OB
      Event_Count : Int;   // Events discarded
   END_VAR
   VAR_TEMP
      erro : Int;
   END_VAR
BEGIN

REGION Network 1: PID do Tanque 1
   // Definição do PID do Tanque 1
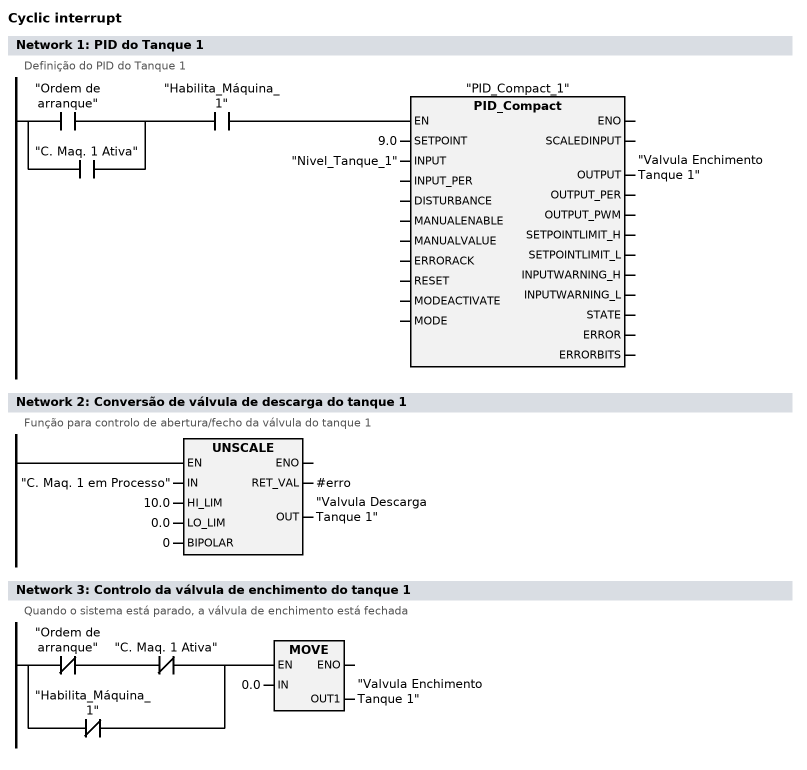
   IF ("Ordem de arranque" OR "C. Maq. 1 Ativa") AND "Habilita_Máquina_1" THEN
       "PID_Compact_1"(Setpoint := 9.0, Input := "Nivel_Tanque_1", Output => "Valvula Enchimento Tanque 1");   // PID_Compact
   END_IF;
END_REGION

REGION Network 2: Conversão de válvula de descarga do tanque 1
   // Função para controlo de abertura/fecho da válvula do tanque 1
   #erro := UNSCALE(IN := "C. Maq. 1 em Processo",
                    HI_LIM := 10.0,
                    LO_LIM := 0.0,
                    BIPOLAR := 0,
                    OUT => "Valvula Descarga Tanque 1");
END_REGION

REGION Network 3: Controlo da válvula de enchimento do tanque 1
   // Quando o sistema está parado, a válvula de enchimento está fechada
   RUNG wire#powerrail
      I_Contact( "Ordem de arranque" )
      I_Contact( "C. Maq. 1 Ativa" )
      wire#w1
      Move(in := 0.0, out1 => "Valvula Enchimento Tanque 1")
   END_RUNG
   RUNG wire#powerrail
      I_Contact( "Habilita_Máquina_1" )
   END_RUNG wire#w1
   // the same network as SCL:
   IF (NOT "Ordem de arranque" AND NOT "C. Maq. 1 Ativa") OR NOT "Habilita_Máquina_1" THEN
       "Valvula Enchimento Tanque 1" := 0.0;
   END_IF;
END_REGION
END_ORGANIZATION_BLOCK

ORGANIZATION_BLOCK "Cyclic interrupt_1"   // OB31, LAD, CyclicInterrupt
TITLE = PID Tanque 2
{ S7_Optimized_Access := 'TRUE' }
VERSION : 0.1
   VAR_INPUT
      Initial_Call : Bool;   // Initial call of this OB
      Event_Count : Int;   // Events discarded
   END_VAR
   VAR_TEMP
      erro : Int;
   END_VAR
BEGIN

REGION Network 1: PID do Tanque 2
   // Definição do PID do Tanque 2
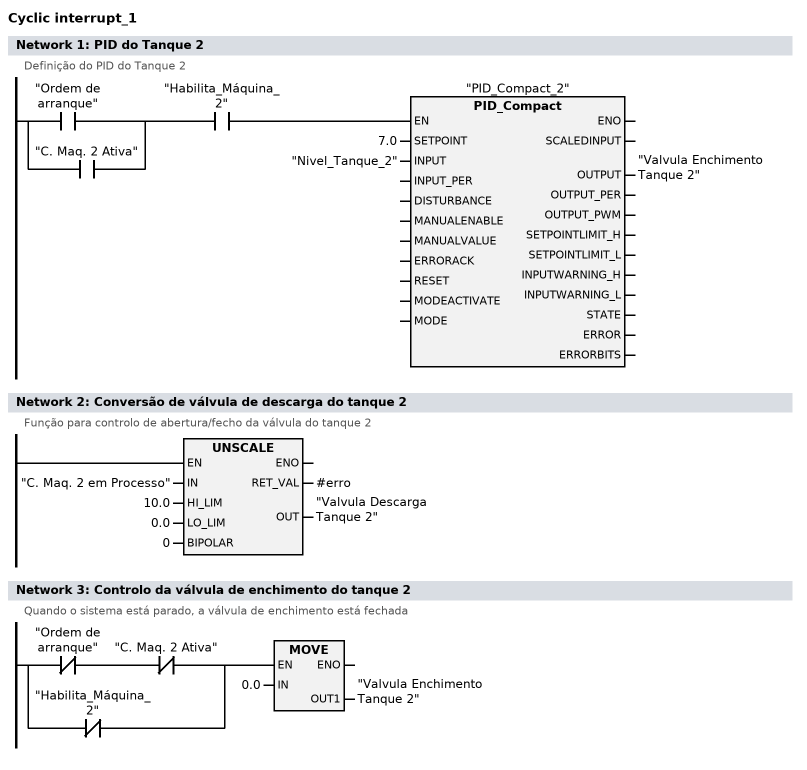
   IF ("Ordem de arranque" OR "C. Maq. 2 Ativa") AND "Habilita_Máquina_2" THEN
       "PID_Compact_2"(Setpoint := 7.0, Input := "Nivel_Tanque_2", Output => "Valvula Enchimento Tanque 2");   // PID_Compact
   END_IF;
END_REGION

REGION Network 2: Conversão de válvula de descarga do tanque 2
   // Função para controlo de abertura/fecho da válvula do tanque 2
   #erro := UNSCALE(IN := "C. Maq. 2 em Processo",
                    HI_LIM := 10.0,
                    LO_LIM := 0.0,
                    BIPOLAR := 0,
                    OUT => "Valvula Descarga Tanque 2");
END_REGION

REGION Network 3: Controlo da válvula de enchimento do tanque 2
   // Quando o sistema está parado, a válvula de enchimento está fechada
   RUNG wire#powerrail
      I_Contact( "Ordem de arranque" )
      I_Contact( "C. Maq. 2 Ativa" )
      wire#w1
      Move(in := 0.0, out1 => "Valvula Enchimento Tanque 2")
   END_RUNG
   RUNG wire#powerrail
      I_Contact( "Habilita_Máquina_2" )
   END_RUNG wire#w1
   // the same network as SCL:
   IF (NOT "Ordem de arranque" AND NOT "C. Maq. 2 Ativa") OR NOT "Habilita_Máquina_2" THEN
       "Valvula Enchimento Tanque 2" := 0.0;
   END_IF;
END_REGION
END_ORGANIZATION_BLOCK

// ===== PLC "PLC_2"  CPU 1512C-1 PN =====

VAR_GLOBAL   // PLC tag table "Default tag table"
   "Clock_Byte" AT %MB500 : Byte;
   "Clock_10Hz" AT %M500.0 : Bool;
   "Clock_5Hz" AT %M500.1 : Bool;
   "Clock_2.5Hz" AT %M500.2 : Bool;
   "Clock_2Hz" AT %M500.3 : Bool;
   "Clock_1.25Hz" AT %M500.4 : Bool;
   "Clock_1Hz" AT %M500.5 : Bool;
   "Clock_0.625Hz" AT %M500.6 : Bool;
   "Clock_0.5Hz" AT %M500.7 : Bool;
END_VAR

DATA_BLOCK "PLC2_Data_Received"   // DB3
{ S7_Optimized_Access := 'FALSE' }
VERSION : 0.1
   VAR
      Contador_Remover_1 : DWord;
      Contador_Remover_2 : DWord;
      Contador_Remover_3 : DWord;
      Contador_Remover_4 : DWord;
      Contador_Remover_5 : DWord;
      Contador_Remover_6 : DWord;
      Contador_Remover_Total : DWord;
      Contador_Máquina_1 : DWord;
      Contador_Máquina_2 : DWord;
      "Valvula Enchimento Tanque 1" : Real;
      "Valvula Descarga Tanque 1" : Real;
      "Valvula Enchimento Tanque 2" : Real;
      "Valvula Descarga Tanque 2" : Real;
      Nivel_1_convertido_Scada : Real;
      Nivel_2_convertido_Scada : Real;
      Aviso_Nenhuma_Máquina_Habilitada : Bool;
      Aviso_Nenhum_Remover_Habilitado : Bool;
      Aviso_Sem_Condições_Empilhar : Bool;
      Set_vel_T3 : Real;
      Set_vel_T4 : Real;
      Set_vel_T6 : Real;
      Set_vel_T5 : Real;
      Set_vel_T7 : Real;
   END_VAR
BEGIN
END_DATA_BLOCK

DATA_BLOCK "PLC2_Data_Sent"   // DB5
{ S7_Optimized_Access := 'FALSE' }
VERSION : 0.1
   VAR
      Start : Bool;
      Stop : Bool;
      Emergência : Bool;
      Habilita_Remover_1 : Bool;
      Habilita_Remover_2 : Bool;
      Habilita_Remover_3 : Bool;
      Habilita_Remover_4 : Bool;
      Habilita_Remover_5 : Bool;
      Habilita_Remover_6 : Bool;
      Habilita_Máquina_1 : Bool;
      Habilita_Máquina_2 : Bool;
      Empilhar : Bool;
      Reset_Cont_Diario : Bool;
      "Reset Contadores Maquinas" : Bool;
      "Reset Contadores Postos" : Bool;
      Máquina1_Tampas : Bool;
      Máquina2_Tampas : Bool;
   END_VAR
BEGIN
END_DATA_BLOCK

// folder: System blocks/Program resources

DATA_BLOCK "PLC_2_Receive_DB"   // DB1
{ S7_Optimized_Access := 'TRUE' }
AUTHOR : SIMATIC
FAMILY : MC7Plus
NAME : TC_IP_v4
VERSION : 1.0
// stored: InstanceOfName TCON_IP_v4
"TCON_IP_v4"
BEGIN
   ID := 1;
   InterfaceId := 64;
   LocalPort := 2000;
   RemoteAddress.ADDR[1] := 192;
   RemoteAddress.ADDR[2] := 168;
   RemoteAddress.ADDR[3] := 228;
   RemoteAddress.ADDR[4] := 231;
END_DATA_BLOCK

DATA_BLOCK "PLC_2_Send_DB"   // DB6
{ S7_Optimized_Access := 'TRUE' }
AUTHOR : SIMATIC
FAMILY : MC7Plus
NAME : TC_IP_v4
VERSION : 1.0
// stored: InstanceOfName TCON_IP_v4
"TCON_IP_v4"
BEGIN
   ID := 2;
   InterfaceId := 64;
   RemotePort := 2000;
   ActiveEstablished := true;
   RemoteAddress.ADDR[1] := 192;
   RemoteAddress.ADDR[2] := 168;
   RemoteAddress.ADDR[3] := 228;
   RemoteAddress.ADDR[4] := 231;
END_DATA_BLOCK

// folder: (top level)

ORGANIZATION_BLOCK "Main"   // OB1, LAD, ProgramCycle
TITLE = "Main Program Sweep (Cycle)"
{ S7_Optimized_Access := 'TRUE' }
VERSION : 0.1
   VAR_INPUT
      Initial_Call : Bool;   // Initial call of this OB
      Remanence : Bool;   // =True, if remanent data are available
   END_VAR
BEGIN

REGION Network 1
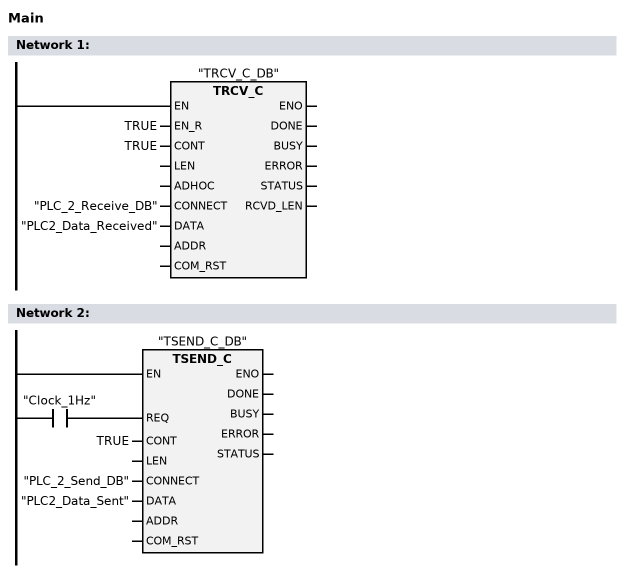
   "TRCV_C_DB"(EN_R := TRUE, CONT := TRUE, CONNECT := "PLC_2_Receive_DB", DATA := "PLC2_Data_Received");   // TRCV_C
END_REGION

REGION Network 2
   "TSEND_C_DB"(REQ := "Clock_1Hz", CONT := TRUE, CONNECT := "PLC_2_Send_DB", DATA := "PLC2_Data_Sent");   // TSEND_C
END_REGION
END_ORGANIZATION_BLOCK

(* ===== HMI "HMI_RT_1" =====
system functions are stored by id; their names below are inferred from use
connection "Connection_1": ETHERNET, S7_1500_OMS
connection "HMI_Connection_1": ETHERNET, S7_1500_OMS

HMI tags "Default tag table"
   "Sensor Tapete 1 Entrada 1" : Bool = PLC "Sensor Tapete 1 Entrada 1" AT %I10.0, 1 s
   "Sensor Tapete 2 Entrada 2" : Bool = PLC "Sensor Tapete 2 Entrada 2" AT %I10.1, 1 s
   "Sensor Inicial Tapete 3 Saida 1" : Bool = PLC "Sensor Inicial Tapete 3 Saida 1" AT %I10.2, 1 s
   "Sensor Final Tapete 3 Saida 1" : Bool = PLC "Sensor Final Tapete 3 Saida 1" AT %I10.3, 1 s
   "Sensor Inicial Tapete 4 Saida 2" : Bool = PLC "Sensor Inicial Tapete 4 Saida 2" AT %I10.4, 1 s
   "Sensor Final Tapete 4 Saida 2" : Bool = PLC "Sensor Final Tapete 4 Saida 2" AT %I10.5, 1 s
   "Sensor Final Tapete 6 Saida 2" : Bool = PLC "Sensor Final Tapete 6 Saida 2" AT %I10.6, 1 s
   "Sensor Final Tapete 7" : Bool = PLC "Sensor Final Tapete 7" AT %I10.7, 1 s
   "Sensor  Grampo Aperto" : Bool = PLC "Sensor  Grampo Aperto" AT %I11.0, 1 s
   "Sensor Posicionador Cima/Baixo" : Bool = PLC "Sensor Posicionador Cima/Baixo" AT %I11.1, 1 s
   "Sensor Posicionador Frente/Tras" : Bool = PLC "Sensor Posicionador Frente/Tras" AT %I11.2, 1 s
   "Sensor Posicionador Presença Peça" : Bool = PLC "Sensor Posicionador Presença Peça" AT %I11.3, 1 s
   "Sensor Saida Posto 1" : Bool = PLC "Sensor Saida Posto 1" AT %I11.4, 100 ms
   "Sensor Saida Posto 2" : Bool = PLC "Sensor Saida Posto 2" AT %I11.5, 100 ms
   "Sensor Saida Posto 3" : Bool = PLC "Sensor Saida Posto 3" AT %I11.6, 100 ms
   "Sensor Saida Posto 4" : Bool = PLC "Sensor Saida Posto 4" AT %I11.7, 100 ms
   "Sensor Saida Posto 5" : Bool = PLC "Sensor Saida Posto 5" AT %I12.0, 100 ms
   "Sensor Saida Posto 6" : Bool = PLC "Sensor Saida Posto 6" AT %I12.1, 100 ms
   "Emissor 1" : Bool = PLC "Emissor 1" AT %Q10.0, 1 s
   "Tapete 1" : Bool = PLC "Tapete 1" AT %Q10.1, 1 s
   "C. Maq. 1 Ativa" : Bool = PLC "C. Maq. 1 Ativa" AT %Q10.2, 1 s
   "C. Maq. 1 Parar" : Bool = PLC "C. Maq. 1 Parar" AT %Q10.3, 1 s
   "C. Maq. 1 Bases/Tampas" : Bool = PLC "C. Maq. 1 Bases/Tampas" AT %Q10.4, 1 s
   "Emissor 2" : Bool = PLC "Emissor 2" AT %Q10.5, 1 s
   "Tapete 2" : Bool = PLC "Tapete 2" AT %Q10.6, 1 s
   "C. Maq. 2 Ativa" : Bool = PLC "C. Maq. 2 Ativa" AT %Q10.7, 1 s
   "C. Maq. 2 Parar" : Bool = PLC "C. Maq. 2 Parar" AT %Q11.0, 1 s
   "C. Maq. 2 Bases/Tampas" : Bool = PLC "C. Maq. 2 Bases/Tampas" AT %Q11.1, 1 s
   "Grampo Aperto" : Bool = PLC "Grampo Aperto" AT %Q11.2, 1 s
   "Grampo Levantar" : Bool = PLC "Grampo Levantar" AT %Q11.3, 1 s
   "Posicionador Cima/Baixo" : Bool = PLC "Posicionador Cima/Baixo" AT %Q11.4, 1 s
   "Posicionador Frente/Tras" : Bool = PLC "Posicionador Frente/Tras" AT %Q11.5, 1 s
   "Posicionador Vacuo" : Bool = PLC "Posicionador Vacuo" AT %Q11.6, 1 s
   "Direcionador 1 Ligar" : Bool = PLC "Direcionador 1 Ligar" AT %Q12.0, 1 s
   "Direcionador 1 Direita" : Bool = PLC "Direcionador 1 Direita" AT %Q12.1, 1 s
   "Direcionador 1 Esquerda" : Bool = PLC "Direcionador 1 Esquerda" AT %Q12.2, 1 s
   "Direcionador 2 Ligar" : Bool = PLC "Direcionador 2 Ligar" AT %Q12.3, 1 s
   "Direcionador 2 Direita" : Bool = PLC "Direcionador 2 Direita" AT %Q12.4, 1 s
   "Direcionador 2 Esquerda" : Bool = PLC "Direcionador 2 Esquerda" AT %Q12.5, 1 s
   "Barreira Posto 3 e 5" : Bool = PLC "Barreira Posto 3 e 5" AT %Q12.6, 1 s
   "Barreira Posto 2 e 4" : Bool = PLC "Barreira Posto 2 e 4" AT %Q12.7, 1 s
   "C. Maq. 1 em Processo" : DInt = PLC "C. Maq. 1 em Processo" AT %ID100, 1 s
   "C. Maq. 2 em Processo" : DInt = PLC "C. Maq. 2 em Processo" AT %ID104, 1 s
   "Nivel Tanque 1" : Real = PLC Nivel_Tanque_1 AT %ID108, 1 s
   "Nivel Tanque 2" : Real = PLC Nivel_Tanque_2 AT %ID112, 1 s
   "Tapete 3" : Real = PLC "Tapete 3" AT %QD100, 1 s
   "Tapete 4" : Real = PLC "Tapete 4" AT %QD104, 1 s
   "Tapete 5" : Real = PLC "Tapete 5" AT %QD108, 1 s
   "Tapete 6" : Real = PLC "Tapete 6" AT %QD112, 1 s
   "Tapete 7" : Real = PLC "Tapete 7" AT %QD116, 1 s
   "Valvula Enchimento Tanque 1" : Real = PLC "Valvula Enchimento Tanque 1" AT %QD120, 1 s
   "Valvula Descarga Tanque 1" : Real = PLC "Valvula Descarga Tanque 1" AT %QD124, 1 s
   "Valvula Enchimento Tanque 2" : Real = PLC "Valvula Enchimento Tanque 2" AT %QD128, 1 s
   "Valvula Descarga Tanque 2" : Real = PLC "Valvula Descarga Tanque 2" AT %QD132, 1 s
   "Contador 1" : DInt = PLC "Contador 1" AT %QD136, 1 s
   "Contador 2" : DInt = PLC "Contador 2" AT %QD140, 1 s
   "Ordem de arranque" : Bool = PLC "Ordem de arranque" AT %M100.0, 1 s
   "Ordem de paragem" : Bool = PLC "Ordem de paragem" AT %M100.1, 1 s
   "M_Tapete1" : Bool = PLC M_Tapete1 AT %M103.0, 1 s
   "M_Tapete2" : Bool = PLC M_Tapete2 AT %M103.1, 1 s
   "M_Tapete3" : Bool = PLC M_Tapete3 AT %M103.2, 1 s
   "M_Tapete4" : Bool = PLC M_Tapete4 AT %M103.3, 1 s
   "M_Tapete5" : Bool = PLC M_Tapete5 AT %M103.4, 1 s
   "M_Tapete6" : Bool = PLC M_Tapete6 AT %M103.5, 1 s
   "M_Tapete7" : Bool = PLC M_Tapete7 AT %M103.6, 1 s
   "V_Tapete3" : Real = PLC V_Tapete3 AT %MD300, 1 s
   "V_Tapete4" : Real = PLC V_Tapete4 AT %MD400, 1 s
   "V_Tapete5" : Real = PLC V_Tapete5 AT %MD500, 1 s
   "V_Tapete6" : Real = PLC V_Tapete6 AT %MD600, 1 s
   "V_Tapete7" : Real = PLC V_Tapete7 AT %MD700, 1 s
   "Etapa_0" : Bool = PLC Etapa_0 AT %M102.7, 1 s
   "Etapa_1" : Bool = PLC Etapa_1 AT %M103.7, 1 s
   "Etapa_2" : Bool = PLC Etapa_2 AT %M104.0, 1 s
   "Etapa_3" : Bool = PLC Etapa_3 AT %M104.1, 1 s
   "Etapa_4" : Bool = PLC Etapa_4 AT %M104.2, 1 s
   "Etapa_5" : Bool = PLC Etapa_5 AT %M104.3, 1 s
   "Etapa_6" : Bool = PLC Etapa_6 AT %M104.4, 1 s
   "Etapa_7" : Bool = PLC Etapa_7 AT %M104.5, 1 s
   "Etapa_8" : Bool = PLC Etapa_8 AT %M104.6, 1 s
   "Etapa_9" : Bool = PLC Etapa_9 AT %M104.7, 1 s
   "Etapa_10" : Bool = PLC Etapa_10 AT %M105.0, 1 s
   "Etapa_11" : Bool = PLC Etapa_11 AT %M105.1, 1 s
   "Etapa_30" : Bool = PLC Etapa_30 AT %M105.2, 1 s
   "Etapa_31" : Bool = PLC Etapa_31 AT %M105.3, 1 s
   "Etapa_32" : Bool = PLC Etapa_32 AT %M105.4, 1 s
   "Etapa_33" : Bool = PLC Etapa_33 AT %M105.5, 1 s
   "Etapa_34" : Bool = PLC Etapa_34 AT %M105.6, 1 s
   "NPosto" : Int = PLC NPosto AT %MW1000, 1 s
   "Etapa_12" : Bool = PLC Etapa_12 AT %M105.7, 1 s
   "Etapa_13" : Bool = PLC Etapa_13 AT %M106.0, 1 s
   "Etapa_14" : Bool = PLC Etapa_14 AT %M106.1, 1 s
   "Etapa_15" : Bool = PLC Etapa_15 AT %M106.2, 1 s
   "Etapa_20" : Bool = PLC Etapa_20 AT %M106.3, 1 s
   "Etapa_35" : Bool = PLC Etapa_35 AT %M106.4, 1 s
   "Etapa_36" : Bool = PLC Etapa_36 AT %M106.5, 1 s
   "Etapa_37" : Bool = PLC Etapa_37 AT %M106.6, 1 s
   "Etapa_38" : Bool = PLC Etapa_38 AT %M106.7, 1 s
   "Etapa_39" : Bool = PLC Etapa_39 AT %M107.0, 1 s
   "Etapa_40" : Bool = PLC Etapa_40 AT %M107.1, 1 s
   "Etapa_50" : Bool = PLC Etapa_50 AT %M107.2, 1 s
   "Empilhar" : Bool = PLC Empilhar AT %M70.0, 1 s
   "Sensor_Geral_Posto" : Bool = PLC Sensor_Geral_Posto AT %M170.0, 1 s
   "Fim de ciclo" : Bool = PLC "Fim de ciclo" AT %M107.5, 1 s
   "Sensor Grampo Levantar" : Bool = PLC "Sensor Grampo Levantar" AT %I12.2, 1 s
   "Entrada_Base" : Bool = PLC Entrada_Base AT %M107.6, 1 s
   "Move Nposto 1" : Bool = PLC "Move Nposto 1" AT %M170.1, 1 s
   "Etapa_100" : Bool = PLC Etapa_100 AT %M150.0, 1 s
   "Etapa_101" : Bool = PLC Etapa_101 AT %M150.1, 1 s
   "Etapa_102" : Bool = PLC Etapa_102 AT %M150.2, 1 s
   "Etapa_103" : Bool = PLC Etapa_103 AT %M150.3, 1 s
   "Etapa_104" : Bool = PLC Etapa_104 AT %M150.4, 1 s
   "Etapa_105" : Bool = PLC Etapa_105 AT %M150.5, 1 s
   "Etapa_106" : Bool = PLC Etapa_106 AT %M150.6, 1 s
   "Etapa_107" : Bool = PLC Etapa_107 AT %M150.7, 1 s
   "Etapa_110" : Bool = PLC Etapa_110 AT %M151.0, 1 s
   "Etapa_111" : Bool = PLC Etapa_111 AT %M151.1, 1 s
   "Etapa_112" : Bool = PLC Etapa_112 AT %M151.2, 1 s
   "Etapa_113" : Bool = PLC Etapa_113 AT %M151.3, 1 s
   "Etapa_114" : Bool = PLC Etapa_114 AT %M151.4, 1 s
   "Etapa_115" : Bool = PLC Etapa_115 AT %M151.5, 1 s
   "Etapa_116" : Bool = PLC Etapa_116 AT %M151.6, 1 s
   "Etapa_117" : Bool = PLC Etapa_117 AT %M151.7, 1 s
   "Etapa_120" : Bool = PLC Etapa_120 AT %M152.0, 1 s
   "Etapa_121" : Bool = PLC Etapa_121 AT %M152.1, 1 s
   "Etapa_122" : Bool = PLC Etapa_122 AT %M152.2, 1 s
   "Etapa_123" : Bool = PLC Etapa_123 AT %M152.3, 1 s
   "Etapa_124" : Bool = PLC Etapa_124 AT %M152.4, 1 s
   "Etapa_125" : Bool = PLC Etapa_125 AT %M152.5, 1 s
   "Etapa_126" : Bool = PLC Etapa_126 AT %M152.6, 1 s
   "Etapa_127" : Bool = PLC Etapa_127 AT %M152.7, 1 s
   "Etapa_130" : Bool = PLC Etapa_130 AT %M153.0, 1 s
   "Etapa_131" : Bool = PLC Etapa_131 AT %M153.1, 1 s
   "Etapa_132" : Bool = PLC Etapa_132 AT %M153.2, 1 s
   "Etapa_133" : Bool = PLC Etapa_133 AT %M153.3, 1 s
   "Etapa_134" : Bool = PLC Etapa_134 AT %M153.4, 1 s
   "Etapa_135" : Bool = PLC Etapa_135 AT %M153.5, 1 s
   "Etapa_136" : Bool = PLC Etapa_136 AT %M153.6, 1 s
   "Etapa_137" : Bool = PLC Etapa_137 AT %M153.7, 1 s
   "Etapa_150" : Bool = PLC Etapa_150 AT %M155.0, 1 s
   "Etapa_151" : Bool = PLC Etapa_151 AT %M155.1, 1 s
   "Etapa_152" : Bool = PLC Etapa_152 AT %M155.2, 1 s
   "Etapa_153" : Bool = PLC Etapa_153 AT %M155.3, 1 s
   "Etapa_154" : Bool = PLC Etapa_154 AT %M155.4, 1 s
   "Etapa_155" : Bool = PLC Etapa_155 AT %M155.5, 1 s
   "Etapa_156" : Bool = PLC Etapa_156 AT %M155.6, 1 s
   "Etapa_157" : Bool = PLC Etapa_157 AT %M155.7, 1 s
   "Pedido_Posic_Ao_Tapete_3" : Bool = PLC Pedido_Posic_Ao_Tapete_3 AT %M160.0, 1 s
   "Pedido_Posic_Ao_Tapete_6" : Bool = PLC Pedido_Posic_Ao_Tapete_6 AT %M160.1, 1 s
   "Pedido_Tap6_Ao_Tapete_4" : Bool = PLC Pedido_Tap6_Ao_Tapete_4 AT %M160.2, 1 s
   "Habilita_Remover_1" : Bool = PLC Habilita_Remover_1 AT %M61.0, 1 s
   "Habilita_Remover_2" : Bool = PLC Habilita_Remover_2 AT %M61.1, 1 s
   "Habilita_Remover_3" : Bool = PLC Habilita_Remover_3 AT %M61.2, 1 s
   "Habilita_Remover_4" : Bool = PLC Habilita_Remover_4 AT %M61.3, 1 s
   "Habilita_Remover_5" : Bool = PLC Habilita_Remover_5 AT %M61.4, 1 s
   "Habilita_Remover_6" : Bool = PLC Habilita_Remover_6 AT %M61.5, 1 s
   "Habilita_Máquina_1" : Bool = PLC Habilita_Máquina_1 AT %M61.6, 1 s
   "Habilita_Máquina_2" : Bool = PLC Habilita_Máquina_2 AT %M61.7, 1 s
   "Máquina1_Tampas" : Bool = PLC Máquina1_Tampas AT %M62.0, 1 s
   "Máquina2_Tampas" : Bool = PLC Máquina2_Tampas AT %M62.1, 1 s
   "Etapa_16" : Bool = PLC Etapa_16 AT %M107.4, 1 s
   "Scan_Estado_31" : Bool = PLC Scan_Estado_31 AT %M165.0, 1 s
   "Contador_Remover_1" : DWord = PLC Contador_Remover_1 AT %MD10, 1 s
   "Contador_Remover_2" : DWord = PLC Contador_Remover_2 AT %MD14, 1 s
   "Contador_Remover_3" : DWord = PLC Contador_Remover_3 AT %MD18, 1 s
   "Contador_Remover_4" : DWord = PLC Contador_Remover_4 AT %MD22, 1 s
   "Contador_Remover_5" : DWord = PLC Contador_Remover_5 AT %MD26, 1 s
   "Contador_Remover_6" : DWord = PLC Contador_Remover_6 AT %MD30, 1 s
   "Start" : Bool = PLC Start AT %M100.2, 1 s
   "Stop" : Bool = PLC Stop AT %M100.3, 1 s
   "Emergência" : Bool = PLC Emergência AT %M180.0, 1 s
   "Reset" : Bool = PLC Reset AT %M100.5, 1 s
   "Aviso_Sem_Condições_Empilhar" : Bool = PLC Aviso_Sem_Condições_Empilhar AT %M154.0, 1 s
   "Aviso_Nenhuma_Máquina_Habilitada" : Bool = PLC Aviso_Nenhuma_Máquina_Habilitada AT %M158.0, 1 s
   "Aviso_Nenhum_Remover_Habilitado" : Bool = PLC Aviso_Nenhum_Remover_Habilitado AT %M162.0, 1 s
   "Contador_Remover_Total" : DWord = PLC Contador_Remover_Total AT %MD34, 1 s
   "Aviso_Sem_Condições_Empilhar(1)" : Int = PLC "Aviso_Sem_Condições_Empilhar(1)" AT %MW154, 1 s
   "Aviso_Nenhuma_Máquina_Habilitada(1)" : Int = PLC "Aviso_Nenhuma_Máquina_Habilitada(1)" AT %MW158, 1 s
   "Aviso_Nenhum_Remover_Habilitado(1)" : Int = PLC "Aviso_Nenhum_Remover_Habilitado(1)" AT %MW162, 1 s
   "Nivel_1_convertido_Scada" : Real = PLC Nivel_1_convertido_Scada AT %ID60, 1 s
   "Contador_Máquina_1" : DWord = PLC Contador_Máquina_1 AT %MD38, 1 s
   "Contador_Máquina_2" : DWord = PLC Contador_Máquina_2 AT %MD42, 1 s
   "Reset Contadores Postos" : Bool = PLC "Reset Contadores Postos" AT %M700.0, 1 s
   "Reset Contadores Maquinas" : Bool = PLC "Reset Contadores Maquinas" AT %M704.0, 1 s
   "Nivel_2_convertido_Scada" : Real = PLC Nivel_2_convertido_Scada AT %ID64, 1 s
   "Emergencia Scada" : Int = PLC "Emergencia Scada" AT %MW166, 1 s
   "Ordem de arranque s ordem paragem" : Bool = PLC "Ordem de arranque s ordem paragem" AT %M100.4, 1 s
   "Name_Login" : WString[254] AT %DB1.DBX0.0
   "Contador_Remover_1_Anterior" : DWord = PLC Contador_Remover_1_Anterior AT %MD310, 1 s
   "Contador_Remover_2_Anterior" : DWord = PLC Contador_Remover_2_Anterior AT %MD314, 1 s
   "Contador_Remover_3_Anterior" : DWord = PLC Contador_Remover_3_Anterior AT %MD318, 1 s
   "Contador_Remover_4_Anterior" : DWord = PLC Contador_Remover_4_Anterior AT %MD322, 1 s
   "Contador_Remover_5_Anterior" : DWord = PLC Contador_Remover_5_Anterior AT %MD326, 1 s
   "Contador_Remover_6_Anterior" : DWord = PLC Contador_Remover_6_Anterior AT %MD330, 1 s
   "Contador_Máquina_1_Anterior" : DWord = PLC Contador_Máquina_1_Anterior AT %MD334, 1 s
   "Contador_Máquina_2_Anterior" : DWord = PLC Contador_Máquina_2_Anterior AT %MD338, 1 s
   "UserName" : WString[30] AT %DB1.DBX0.0

analog alarms
   1: 'Aviso_Sem_Condições_Empilhar', class Errors, trigger "Aviso_Sem_Condições_Empilhar(1)"
   2: 'Aviso_Nenhuma_Máquina_Habilitada', class Errors, trigger "Aviso_Nenhuma_Máquina_Habilitada(1)"
   3: 'Aviso_Nenhum_Remover_Habilitado', class Errors, trigger "Aviso_Nenhum_Remover_Habilitado(1)"
   4: 'Alarme Botão de Emergencia', class Errors, trigger "Emergencia Scada"

text list "Start_stop": 0 'Start'; 1 'Stop'

screen "Event" 1024x690
   GraphicView "Graphic view_1" at 7,6 size 640x680; Picture "Captura de ecrã 2024-12-14 002524"
   Rectangle "Template_Rectangle_1" at 453,137 size 24x56
      Appearance <- "Tapete 2"
   Rectangle "Template_Rectangle_2" at 453,119 size 24x17
      Appearance <- "Emissor 2"
   TextField "Template_Text field_1" at 461,144 size 12x37; Text 'Tapete 2'
   Circle "Circle_5" at 558,102 size 26x26
      Appearance <- "Valvula Enchimento Tanque 2"
   Rectangle "Template_Rectangle_15" at 207,137 size 24x55
      Appearance <- "Tapete 1"
   Circle "Circle_2" at 270,102 size 26x26
      Appearance <- "Valvula Enchimento Tanque 1"
   Rectangle "Template_Rectangle_17" at 207,119 size 24x17
      Appearance <- "Emissor 1"
   TextField "Template_Text field_9" at 215,143 size 12x37; Text 'Tapete 1'
   Circle "Circle_6" at 558,151 size 26x26
      Appearance <- "C. Maq. 2 em Processo"
   Rectangle "Rectangle_3" at 569,246 size 20x28
      Appearance <- "C. Maq. 2 em Processo"
   Rectangle "Rectangle_4" at 296,246 size 21x28
      Appearance <- "C. Maq. 1 em Processo"
   Circle "Circle_4" at 173,283 size 20x20
      Appearance <- "C. Maq. 1 Ativa"
   Rectangle "Template_Rectangle_11" at 353,410 size 132x26
      Appearance <- "Tapete 5"
   Rectangle "Template_Rectangle_13" at 459,353 size 26x57
      Appearance <- "Tapete 4"
   TextField "Template_Text field_11" at 467,358 size 13x47; Text 'Tapete 4'
   TextField "Template_Text field_14" at 385,414 size 56x16; Text 'Tapete 5'
   Rectangle "Template_Rectangle_12" at 194,353 size 25x58
      Appearance <- "Tapete 3"
   TextField "Template_Text field_8" at 203,356 size 13x47; Text 'Tapete 3'
   Rectangle "Template_Rectangle_5" at 194,410 size 25x128
      Appearance <- "Tapete 7"
   IOField "Template_I/O field_6" at 194,602 size 24x14; FormatPattern 999
      ProcessValue <- "Contador_Remover_1"
   TextField "Template_Text field_7" at 298,524 size 14x23; Text 'Text'
   TextField "Template_Text field_13" at 199,449 size 16x56; Text 'Tapete 7'
   Rectangle "Template_Rectangle_9" at 219,410 size 136x26
      Appearance <- "Tapete 6"
   TextField "Template_Text field_12" at 259,415 size 56x16; Text 'Tapete 6'
   Rectangle "Template_Rectangle_3" at 120,436 size 27x64
      Appearance <- "Sensor Saida Posto 2"
   Rectangle "Template_Rectangle_4" at 157,538 size 27x61
      Appearance <- "Sensor Saida Posto 5"
   Rectangle "Template_Rectangle_6" at 120,538 size 27x61
      Appearance <- "Sensor Saida Posto 4"
   TextField "Template_Text field_4" at 129,545 size 13x48; Text 'POSTO 4'
   TextField "Template_Text field_5" at 166,547 size 13x48; Text 'POSTO 5'
   IOField "Template_I/O field_2" at 158,423 size 24x12; FormatPattern 999
      ProcessValue <- "Contador_Remover_3"
   IOField "Template_I/O field_4" at 158,602 size 24x14; FormatPattern 999
      ProcessValue <- "Contador_Remover_5"
   IOField "Template_I/O field_5" at 122,602 size 24x14; FormatPattern 999
      ProcessValue <- "Contador_Remover_4"
   Rectangle "Template_Rectangle_7" at 51,505 size 64x30
      Appearance <- "Sensor Saida Posto 6"
   TextField "Template_Text field_6" at 60,513 size 48x13; Text 'POSTO 6'
   IOField "Template_I/O field_3" at 22,513 size 26x12; FormatPattern 999
      ProcessValue <- "Contador_Remover_6"
   Rectangle "Template_Rectangle_14" at 115,500 size 6x38
      Appearance <- "Barreira Posto 2 e 4"
   Rectangle "Template_Rectangle_16" at 157,436 size 27x64
      Appearance <- "Sensor Saida Posto 3"
   TextField "Template_Text field_10" at 129,444 size 13x48; Text 'POSTO 2'
   IOField "Template_I/O field_1" at 122,423 size 23x13; FormatPattern 999
      ProcessValue <- "Contador_Remover_2"
   Circle "Circle_3" at 427,282 size 20x20
      Appearance <- "C. Maq. 2 Ativa"
   Rectangle "Template_Rectangle_18" at 194,538 size 25x61
      Appearance <- "Sensor Saida Posto 1"
   TextField "Text field_12" at 18,4 size 146x22; Text 'Nenhuma Máquina'
      Visibility <- "Aviso_Nenhuma_Máquina_Habilitada"
   TextField "Text field_13" at 18,71 size 116x22; Text 'Nenhum Posto'
      Visibility <- "Aviso_Nenhum_Remover_Habilitado"
   TextField "Text field_14" at 18,142 size 119x22; Text 'Sem condições'
      Visibility <- "Aviso_Sem_Condições_Empilhar"
   TextField "Template_Text field_3" at 202,548 size 13x48; Text 'POSTO 1'
   TextField "Template_Text field_2" at 165,444 size 13x48; Text 'POSTO 3'
   Rectangle "Template_Rectangle_8" at 152,500 size 6x38
      Appearance <- "Barreira Posto 3 e 5"
   Bar "Bar_1" at 322,23 size 41x157; MinimumValue 0; MaximumValue 300
      ProcessValue <- "Nivel_1_convertido_Scada"
   Bar "Bar_2" at 607,23 size 39x157; MinimumValue 0; MaximumValue 300
      ProcessValue <- "Nivel_2_convertido_Scada"
   IOField "I/O field_9" at 246,64 size 65x32; FormatPattern 999
      ProcessValue <- "Nivel_1_convertido_Scada"
   IOField "I/O field_1" at 540,64 size 62x32; FormatPattern 999
      ProcessValue <- "Nivel_2_convertido_Scada"
   IOField "Template_I/O field_7" at 278,602 size 89x27; FormatPattern 999
      ProcessValue <- "Contador_Remover_Total"
   TextField "Template_Text field_15" at 276,583 size 95x16; Text 'Contador Total'
   TextField "Text field_15" at 19,159 size 109x22; Text 'para empilhar'
      Visibility <- "Aviso_Sem_Condições_Empilhar"
   TextField "Text field_16" at 18,26 size 82x22; Text 'Habilitada'
      Visibility <- "Aviso_Nenhuma_Máquina_Habilitada"
   TextField "Text field_17" at 18,94 size 82x22; Text 'Habilitado'
      Visibility <- "Aviso_Nenhum_Remover_Habilitado"
   Button "Button_7" at 679,267 size 312x61; TextOff 'Habilitar/Remover Postos'; TextOn 'Pop-up screen_1'
      on Click: function_efd93a16("Habilitar/Remover Postos", 648, 418, -1, -1, 1)
   Button "Button_1" at 677,107 size 308x65; TextOff 'Habilitar/Remover Máquinas'
      on Click: function_efd93a16("Habilitar/Remover Máquinas", 648, 418, -1, -1, 1)
   Button "Button_2" at 677,184 size 310x68; TextOff 'Habilitar/Remover Tipos Processos'
      on Click: function_efd93a16("Habilitar/Remover Tipos Processos", 648, 418, -1, -1, 1)
   GraphicView "Graphic view_2" at 649,342 size 373x346; Picture "Graphic_92"
   Button "Button_14" at 863,19 size 115x65; TextOff 'EMERGENCIA'
      on Press: InvertBit("Emergência")
      Appearance <- "Emergência"
   Button "Button_8" at 685,28 size 61x49; TextOff 'START'
      on Release: ResetBit("Start")
      on Press: SetBit("Start")
      Appearance <- "Ordem de arranque s ordem paragem"
   Button "Button_5" at 772,28 size 61x50; TextOff 'STOP'
      on Release: SetBit("Stop")
      on Press: ResetBit("Stop")
      Appearance <- "Ordem de paragem"
   IOField "Template_I/O field_8" at 296,275 size 21x16; FormatPattern 999
      ProcessValue <- "Contador_Máquina_1"
   IOField "Template_I/O field_9" at 569,276 size 21x16; FormatPattern 999
      ProcessValue <- "Contador_Máquina_2"
   TextField "Text field_51" at 288,68 size 14x22; Text 'L'
   TextField "Text field_1" at 580,68 size 14x22; Text 'L'
   TextField "Text field_52" at 266,513 size 371x70; Text 'ATENÇÃO! EMERGÊNCIA PRESSIONADA'
      Visibility <- "Emergência"
   Circle "Circle_1" at 270,151 size 26x26
      Appearance <- "C. Maq. 1 em Processo"

screen "Home" 1024x690
   TextField "Text field_1" at 515,149 size 38x62; Text 'Text'
   GraphicView "Graphic view_1" at 1,1 size 1023x683; Picture "Graphic_89"
   TextField "Text field_5" at 560,533 size 383x82; Text 'Automatização de um Sistema de Maquinação'
   TextField "Text field_6" at 553,616 size 380x27; Text 'Para aceder, inicie previamente sessão'
   TextField "Text field_52" at 205,395 size 404x76; Text 'ATENÇÃO! EMERGÊNCIA PRESSIONADA'
      Visibility <- "Emergência"
   TextField "Text field_2" at 813,167 size 110x42; Text '2222804'
   TextField "Text field_3" at 814,246 size 119x42; Text '2222007'
   TextField "Text field_4" at 772,131 size 189x42; Text 'Bruna Sousa'
   TextField "Text field_7" at 772,211 size 188x42; Text 'Flávio Duarte'

screen "Alarm" 1024x690
   GraphicView "Graphic view_1" at 1,2 size 1023x686; Picture "Graphic_89"
   TextField "Text field_30" at 251,0 size 230x39; Text 'Alarmes ativos'
   TextField "Text field_5" at 216,314 size 305x39; Text 'Histórico de alarmes'
   AlarmView "Alarm view_2" at 79,38 size 581x280
   AlarmView "Alarm view_1" at 79,352 size 581x284; AlarmLog "Alarm_log_1"
   TextField "Text field_52" at 728,134 size 289x56; Text 'ATENÇÃO! EMERGÊNCIA PRESSIONADA'
      Visibility <- "Emergência"

screen "Maintenance" 1024x690
   GraphicView "Graphic view_1" at 1,1 size 1023x684; Picture "Graphic_89"
   Button "Button_1" at 786,140 size 192x32; TextOff 'Contadores'; TextOn 'contadores'
      on Click: function_efd93a16("Contadores", 649, 418, -1, -1, 1)
   Button "Button_2" at 786,184 size 192x32; TextOff 'Contadores Maquinas'; TextOn 'contadores Maquinas'
      on Click: function_efd93a16("Contadores Maquinas", 649, 418, -1, -1, 1)
   Button "Button_3" at 786,227 size 193x32; TextOff 'Reset Cont. Postos'
      Appearance <- "Reset Contadores Postos"
      ObjectEnable <- "Reset Contadores Postos"
      on Release: ResetBit("Reset Contadores Postos")
      on Press: SetBit("Reset Contadores Postos")
   Button "Button_5" at 786,271 size 193x32; TextOff 'Reset Cont. Maquinas'
      on Release: ResetBit("Reset Contadores Maquinas")
      on Press: SetBit("Reset Contadores Maquinas")
      Appearance <- "Reset Contadores Maquinas"
   TextField "Text field_52" at 205,395 size 404x76; Text 'ATENÇÃO! EMERGÊNCIA PRESSIONADA'
      Visibility <- "Emergência"

screen "Trends" 1024x690
   GraphicView "Graphic view_1" at 1,3 size 1022x682; Picture "Graphic_89"
   Button "Button_1" at 783,154 size 192x32; TextOff 'Nível 1'; TextOn 'Nível'
      on Click: function_efd93a16("Nível 1", 0, 214, -1, -1, 1)
   Button "Button_2" at 783,198 size 192x32; TextOff 'Nível 2'
      on Click: function_efd93a16("Nível 2", 0, 214, -1, -1, 1)
   Button "Button_3" at 783,245 size 192x32; TextOff 'Nível 1 VS Nível 2'; TextOn 'Potência'
      on Click: function_efd93a16("Nível 1 VS Nível 2", 0, 214, -1, -1, 1)
   TextField "Text field_52" at 205,395 size 404x76; Text 'ATENÇÃO! EMERGÊNCIA PRESSIONADA'
      Visibility <- "Emergência"
   Button "Button_4" at 783,291 size 192x32; TextOff 'Maquina 1 Processo'
      on Click: function_efd93a16("Maquina 1 Processo", 0, 214, -1, -1, 1)
   Button "Button_5" at 783,336 size 192x32; TextOff 'Maquina 2 Processo'
      on Click: function_efd93a16("Maquina 2 Processo", 0, 214, -1, -1, 1)
   Button "Button_6" at 783,382 size 192x32; TextOff 'Tapete 3'; TextOn 'Tapetes'
      on Click: function_efd93a16("Tapete 3", 0, 214, -1, -1, 1)
   Button "Button_7" at 783,426 size 192x32; TextOff 'Tapete 4'
      on Click: function_efd93a16("Tapete 4", 0, 214, -1, -1, 1)
   Button "Button_8" at 783,471 size 192x32; TextOff 'Tapete 5'
      on Click: function_efd93a16("Tapete 5", 0, 214, -1, -1, 1)
   Button "Button_9" at 783,517 size 192x32; TextOff 'Tapete 6'
      on Click: function_efd93a16("Tapete 6", 0, 214, -1, -1, 1)
   Button "Button_10" at 783,565 size 192x32; TextOff 'Tapete 7'
      on Click: function_efd93a16("Tapete 7", 0, 214, -1, -1, 1)

PopupScreen "Habilitar/Remover Postos" 375x350
   Button "Button_4" at 189,90 size 46x37; TextOff 'P1'
      on Press: InvertBit("Habilita_Remover_1")
      Appearance <- "Habilita_Remover_1"
   Button "Button_5" at 189,130 size 46x37; TextOff 'P2'
      on Press: InvertBit("Habilita_Remover_2")
      Appearance <- "Habilita_Remover_2"
   Button "Button_6" at 189,170 size 46x37; TextOff 'P3'
      on Press: InvertBit("Habilita_Remover_3")
      Appearance <- "Habilita_Remover_3"
   Button "Button_9" at 189,210 size 46x37; TextOff 'P4'
      on Press: InvertBit("Habilita_Remover_4")
      Appearance <- "Habilita_Remover_4"
   Button "Button_10" at 189,250 size 45x36; TextOff 'P5'
      on Press: InvertBit("Habilita_Remover_5")
      Appearance <- "Habilita_Remover_5"
   Button "Button_11" at 189,290 size 45x37; TextOff 'P6'
      on Press: InvertBit("Habilita_Remover_6")
      Appearance <- "Habilita_Remover_6"
   GraphicView "Graphic view_1" at 252,11 size 101x319; Picture "Graphic_97"
   TextField "Text field_1" at 23,17 size 224x29; Text 'Habilitar # Remover'
   TextField "Text field_9" at 70,93 size 84x29; Text 'Posto 1'
   TextField "Text field_2" at 70,132 size 84x29; Text 'Posto 2'
   TextField "Text field_3" at 70,171 size 84x29; Text 'Posto 3'
   TextField "Text field_4" at 70,211 size 84x29; Text 'Posto 4'
   TextField "Text field_5" at 70,253 size 84x29; Text 'Posto 5'
   TextField "Text field_6" at 70,293 size 84x29; Text 'Posto 6'
   TextField "Text field_7" at 89,47 size 76x29; Text 'Postos'

PopupScreen "Habilitar/Remover Máquinas" 375x350
   Button "Button_1" at 60,81 size 70x47; TextOff 'M1'
      on Press: InvertBit("Habilita_Máquina_1")
      Appearance <- "Habilita_Máquina_1"
      ObjectEnable <- "Ordem de arranque"
   TextField "Text field_9" at 13,22 size 158x22; Text 'Habilitar # Remover'
   Button "Button_2" at 60,237 size 69x47; TextOff 'M2'
      on Press: InvertBit("Habilita_Máquina_2")
      Appearance <- "Habilita_Máquina_2"
      ObjectEnable <- "Ordem de arranque"
   GraphicView "Graphic view_1" at 180,18 size 182x147; Picture "Graphic_94"
   GraphicView "Graphic view_2" at 180,182 size 182x147; Picture "Graphic_94"
   TextField "Text field_2" at 54,46 size 82x22; Text 'Máquina 1'
   TextField "Text field_1" at 13,182 size 158x22; Text 'Habilitar # Remover'
   TextField "Text field_3" at 56,204 size 82x22; Text 'Máquina 2'

PopupScreen "Habilitar/Remover Tipos Processos" 375x350
   Button "Button_12" at 182,172 size 49x45; TextOff 'M1'
      on Press: InvertBit("Máquina1_Tampas")
      Appearance <- "Máquina1_Tampas"
      ObjectEnable <- "Ordem de arranque"
   TextField "Text field_10" at 23,184 size 143x22; Text 'Máquina 1 Tampas'
   Button "Button_13" at 182,258 size 49x45; TextOff 'M2'
      on Press: InvertBit("Máquina2_Tampas")
      Appearance <- "Máquina2_Tampas"
      ObjectEnable <- "Ordem de arranque"
   TextField "Text field_11" at 23,268 size 143x22; Text 'Máquina 2 Tampas'
   TextField "Text field_2" at 31,56 size 115x22; Text 'Habilitar Modo'
   Button "Button_3" at 182,56 size 49x45; TextOff 'CX'
      on Press: InvertBit("Empilhar")
      Appearance <- "Empilhar"
      ObjectEnable <- "Ordem de arranque"
   GraphicView "Graphic view_1" at 243,160 size 85x70; Picture "Graphic_98"
   GraphicView "Graphic view_2" at 243,246 size 85x70; Picture "Graphic_98"
   GraphicView "Graphic view_3" at 244,39 size 85x39; Picture "Graphic_98"
   GraphicView "Graphic view_4" at 244,78 size 84x41; Picture "Graphic_99"
   TextField "Text field_1" at 23,84 size 144x22; Text 'Caixas Empilhadas'

PopupScreen "Contadores" 375x350
   IOField "Template_I/O field_6" at 113,93 size 53x31; FormatPattern 999
      ProcessValue <- "Contador_Remover_1"
   IOField "Template_I/O field_4" at 113,253 size 54x31; FormatPattern 999
      ProcessValue <- "Contador_Remover_5"
   IOField "Template_I/O field_5" at 113,213 size 53x28; FormatPattern 999
      ProcessValue <- "Contador_Remover_4"
   IOField "Template_I/O field_3" at 113,293 size 54x29; FormatPattern 999
      ProcessValue <- "Contador_Remover_6"
   IOField "Template_I/O field_1" at 113,133 size 53x29; FormatPattern 999
      ProcessValue <- "Contador_Remover_2"
   IOField "Template_I/O field_2" at 113,173 size 54x28; FormatPattern 999
      ProcessValue <- "Contador_Remover_3"
   TextField "Text field_9" at 19,93 size 84x29; Text 'Posto 1'
   TextField "Text field_1" at 19,132 size 84x29; Text 'Posto 2'
   TextField "Text field_2" at 19,171 size 84x29; Text 'Posto 3'
   TextField "Text field_3" at 19,211 size 84x29; Text 'Posto 4'
   TextField "Text field_4" at 19,253 size 84x29; Text 'Posto 5'
   TextField "Text field_5" at 19,293 size 84x29; Text 'Posto 6'
   GraphicView "Graphic view_1" at 252,11 size 101x319; Picture "Graphic_97"
   TextField "Text field_6" at 66,6 size 125x29; Text 'Contadores'
   TextField "Text field_7" at 90,35 size 76x29; Text 'Postos'
   IOField "Template_I/O field_7" at 182,93 size 53x31; FormatPattern 999
      ProcessValue <- "Contador_Remover_1_Anterior"
   IOField "Template_I/O field_8" at 182,253 size 54x31; FormatPattern 999
      ProcessValue <- "Contador_Remover_5_Anterior"
   IOField "Template_I/O field_9" at 182,213 size 53x28; FormatPattern 999
      ProcessValue <- "Contador_Remover_4_Anterior"
   IOField "Template_I/O field_10" at 182,293 size 54x29; FormatPattern 999
      ProcessValue <- "Contador_Remover_6_Anterior"
   IOField "Template_I/O field_11" at 182,133 size 53x29; FormatPattern 999
      ProcessValue <- "Contador_Remover_2_Anterior"
   IOField "Template_I/O field_12" at 182,173 size 54x28; FormatPattern 999
      ProcessValue <- "Contador_Remover_3_Anterior"
   TextField "Text field_8" at 110,71 size 49x23; Text 'Atual'
   TextField "Text field_10" at 172,72 size 73x23; Text 'Anterior'

PopupScreen "Contadores Maquinas" 375x350
   IOField "Template_I/O field_8" at 94,68 size 63x24; FormatPattern 999
      ProcessValue <- "Contador_Máquina_1"
   GraphicView "Graphic view_1" at 167,15 size 182x147; Picture "Graphic_94"
   GraphicView "Graphic view_2" at 167,179 size 182x147; Picture "Graphic_94"
   TextField "Text field_3" at 29,24 size 114x29; Text 'Máquina 1'
   TextField "Text field_1" at 29,180 size 114x29; Text 'Máquina 2'
   TextField "Text field_8" at 36,68 size 49x23; Text 'Atual'
   TextField "Text field_10" at 13,102 size 73x23; Text 'Anterior'
   IOField "Template_I/O field_1" at 94,102 size 63x24; FormatPattern 999
      ProcessValue <- "Contador_Máquina_1_Anterior"
   IOField "Template_I/O field_2" at 96,231 size 63x24; FormatPattern 999
      ProcessValue <- "Contador_Máquina_2"
   TextField "Text field_2" at 38,231 size 49x23; Text 'Atual'
   TextField "Text field_4" at 15,265 size 73x23; Text 'Anterior'
   IOField "Template_I/O field_3" at 96,265 size 63x24; FormatPattern 999
      ProcessValue <- "Contador_Máquina_2_Anterior"

PopupScreen "Nível 1" 778x554
   TrendView "Nível" at 3,4 size 773x544

PopupScreen "Nível 2" 778x554
   TrendView "Nível" at 3,0 size 773x550

PopupScreen "Nível 1 VS Nível 2" 778x554
   TrendView "Nível" at 3,0 size 773x550

PopupScreen "Maquina 1 Processo" 778x554
   TrendView "Nível" at 3,4 size 773x544

PopupScreen "Maquina 2 Processo" 778x554
   TrendView "Nível" at 3,4 size 773x544

PopupScreen "Tapete 3" 778x554
   TrendView "Nível" at 3,4 size 773x544

PopupScreen "Tapete 4" 778x554
   TrendView "Nível" at 3,7 size 771x540

PopupScreen "Tapete 5" 778x554
   TrendView "Nível" at 3,5 size 771x543

PopupScreen "Tapete 6" 778x554
   TrendView "Nível" at 3,4 size 773x544

PopupScreen "Tapete 7" 778x554
   TrendView "Nível" at 3,4 size 773x544

scheduled task "Produção"
   on Action: function_fd03fc5c("Report_Diario")

scheduled task "User"
   on Action: function_f41c6f6c("UserName")
*)